KUKA KRL program: MyProgram_065().src

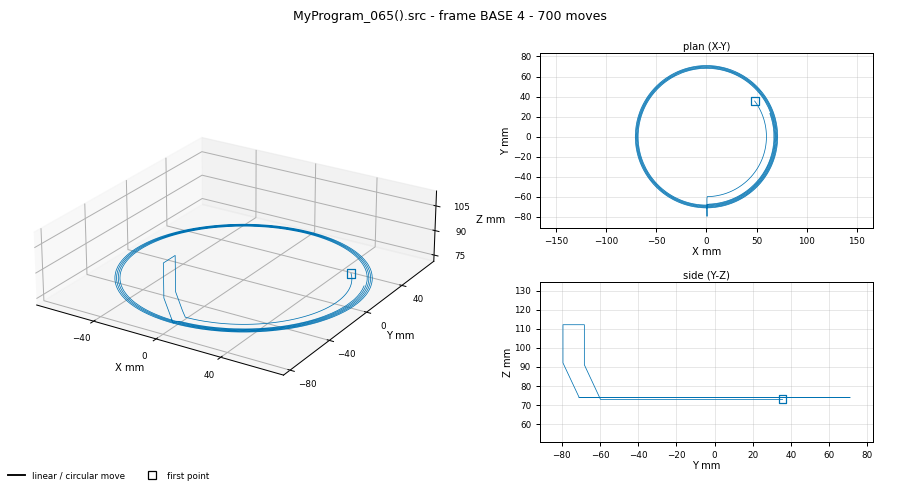
[picture p0: tool path of MyProgram_065().src in frame BASE 4, 700 of 700 moves have a stored position in this frame; points joined in program order, loops and branches not executed]
&ACCESS RVP
&REL 1
&PARAM TEMPLATE = C:\KRC\Roboter\Template\vorgabe
&PARAM EDITMASK = *
DEF MyProgram_065()
; ---- Setting reference (Base) ----
$BASE = BASE_DATA[4]

; --------------------------
; ---- Setting tool (TCP) ----
$TOOL = TOOL_DATA[3]
; --------------------------

$VEL.CP = VEL_APROX_PRINT
Startdeposition()
$VEL.CP = VEL_PRINT
LIN {X 47.9993,Y 35.5944,Z 73,A 29.5508,B 24.867,C -2.6616,E1 25.1296,E2 54.3214} C_DIS
LIN {X 49.6814,Y 33.206,Z 73,A 26.7608,B 24.8676,C -2.6549,E1 25.134,E2 57.1135} C_DIS
LIN {X 51.2611,Y 30.7113,Z 73,A 23.9498,B 24.8683,C -2.648,E1 25.1381,E2 59.9264} C_DIS
LIN {X 52.7031,Y 28.165,Z 73,A 21.1603,B 24.869,C -2.6409,E1 25.1419,E2 62.7181} C_DIS
LIN {X 54.019,Y 25.5508,Z 73,A 18.3589,B 24.8698,C -2.6333,E1 25.1453,E2 65.5225} C_DIS
LIN {X 55.2106,Y 22.862,Z 73,A 15.5717,B 24.8705,C -2.6261,E1 25.1484,E2 68.3114} C_DIS
LIN {X 56.2606,Y 20.1403,Z 73,A 12.7899,B 24.8713,C -2.6184,E1 25.1511,E2 71.096} C_DIS
LIN {X 57.1824,Y 17.3512,Z 73,A 9.9851,B 24.8721,C -2.6104,E1 25.1535,E2 73.9038} C_DIS
LIN {X 57.9667,Y 14.5172,Z 73,A 7.1908,B 24.8728,C -2.6025,E1 25.1555,E2 76.7007} C_DIS
LIN {X 58.6083,Y 11.6601,Z 73,A 4.4011,B 24.8736,C -2.5944,E1 25.1571,E2 79.4934} C_DIS
LIN {X 59.1091,Y 8.7751,Z 73,A 1.6072,B 24.8744,C -2.586,E1 25.1583,E2 82.2905} C_DIS
LIN {X 59.4694,Y 5.855,Z 73,A -1.1879,B 24.8752,C -2.5779,E1 25.1592,E2 85.0884} C_DIS
LIN {X 59.6848,Y 2.935,Z 73,A -3.9767,B 24.8761,C -2.5695,E1 25.1597,E2 87.8804} C_DIS
LIN {X 59.7559,Y 0.0054,Z 73,A -6.7286,B 24.8768,C -2.562,E1 25.1597,E2 90.6337} C_DIS
LIN {X 59.6838,Y -2.9525,Z 73,A -9.5735,B 24.8777,C -2.5528,E1 25.1595,E2 93.4834} C_DIS
LIN {X 59.4691,Y -5.8582,Z 73,A -12.3571,B 24.8785,C -2.5442,E1 25.1588,E2 96.2709} C_DIS
LIN {X 59.1109,Y -8.7628,Z 73,A -15.1438,B 24.8793,C -2.5358,E1 25.1578,E2 99.061} C_DIS
LIN {X 58.611,Y -11.6459,Z 73,A -17.9348,B 24.8801,C -2.5273,E1 25.1563,E2 101.8557} C_DIS
LIN {X 57.9566,Y -14.5566,Z 73,A -20.7653,B 24.8809,C -2.5191,E1 25.1545,E2 104.6892} C_DIS
LIN {X 57.1775,Y -17.3669,Z 73,A -23.5438,B 24.8817,C -2.5109,E1 25.1524,E2 107.4714} C_DIS
LIN {X 56.2608,Y -20.1398,Z 73,A -26.3255,B 24.8824,C -2.5027,E1 25.1498,E2 110.2566} C_DIS
LIN {X 55.2091,Y -22.8658,Z 73,A -29.1109,B 24.8832,C -2.4946,E1 25.1469,E2 113.0457} C_DIS
LIN {X 54.0255,Y -25.5368,Z 73,A -31.8935,B 24.8839,C -2.4868,E1 25.1437,E2 115.8317} C_DIS
LIN {X 52.7131,Y -28.1462,Z 73,A -34.6833,B 24.8847,C -2.4789,E1 25.1401,E2 118.6255} C_DIS
LIN {X 51.2479,Y -30.7332,Z 73,A -37.5078,B 24.8854,C -2.4714,E1 25.1361,E2 121.4531} C_DIS
LIN {X 49.6819,Y -33.2053,Z 73,A -40.2967,B 24.886,C -2.464,E1 25.1319,E2 124.2455} C_DIS
LIN {X 47.9963,Y -35.5983,Z 73,A -43.0873,B 24.8867,C -2.4568,E1 25.1273,E2 127.0396} C_DIS
LIN {X 46.1955,Y -37.906,Z 73,A -45.8892,B 24.8874,C -2.4496,E1 25.1224,E2 129.8455} C_DIS
LIN {X 44.2702,Y -40.1376,Z 73,A -48.6868,B 24.888,C -2.4432,E1 25.1172,E2 132.6458} C_DIS
LIN {X 42.2524,Y -42.2566,Z 73,A -51.4776,B 24.8886,C -2.4367,E1 25.1118,E2 135.4399} C_DIS
LIN {X 40.133,Y -44.2745,Z 73,A -54.2703,B 24.8891,C -2.4305,E1 25.1061,E2 138.2359} C_DIS
LIN {X 37.9019,Y -46.1988,Z 73,A -57.0803,B 24.8897,C -2.4246,E1 25.1001,E2 141.049} C_DIS
LIN {X 35.5942,Y -47.9994,Z 73,A -59.8738,B 24.8902,C -2.419,E1 25.0939,E2 143.8456} C_DIS
LIN {X 33.2009,Y -49.6849,Z 73,A -62.6695,B 24.8907,C -2.4137,E1 25.0874,E2 146.6443} C_DIS
LIN {X 30.728,Y -51.2511,Z 73,A -65.4647,B 24.8911,C -2.4088,E1 25.0808,E2 149.4424} C_DIS
LIN {X 28.1363,Y -52.7183,Z 73,A -68.3046,B 24.8915,C -2.4042,E1 25.0738,E2 152.2848} C_DIS
LIN {X 25.5294,Y -54.0289,Z 73,A -71.094,B 24.8919,C -2.3999,E1 25.0668,E2 155.0769} C_DIS
LIN {X 22.858,Y -55.2123,Z 73,A -73.8869,B 24.8923,C -2.396,E1 25.0596,E2 157.8725} C_DIS
LIN {X 20.1306,Y -56.2641,Z 73,A -76.6835,B 24.8926,C -2.3925,E1 25.0523,E2 160.6715} C_DIS
LIN {X 17.3549,Y -57.1812,Z 73,A -79.4798,B 24.8929,C -2.3893,E1 25.0449,E2 163.4701} C_DIS
LIN {X 14.236,Y -58.0353,Z 73,A -81.964,B 24.8919,C -2.3996,E1 25.0382,E2 165.926} C_DIS
LIN {X 11.905,Y -58.558,Z 73,A -84.7921,B 24.8932,C -2.3859,E1 25.0304,E2 168.783} C_DIS
LIN {X 9.482,Y -58.9998,Z 73,A -87.2165,B 24.8935,C -2.3827,E1 25.0238,E2 171.2124} C_DIS
LIN {X 6.5815,Y -59.3934,Z 73,A -90.0194,B 24.8936,C -2.3811,E1 25.016,E2 174.017} C_DIS
LIN {X 3.6648,Y -59.6444,Z 73,A -92.8251,B 24.8937,C -2.3798,E1 25.0082,E2 176.8243} C_DIS
LIN {X 0.7394,Y -59.7523,Z 73,A -95.6385,B 24.8938,C -2.3788,E1 25.0003,E2 179.6396} C_DIS
LIN {X 0.7394,Y -59.7523,Z 73,A -95.6385,B 24.8938,C -2.3788,E1 25.0003,E2 179.6396} C_DIS
Enddeposition()
LIN {X 0.4348,Y -61.8654,Z 77.5315,A -95.642,B 24.8937,C -2.3803,E1 25.0003,E2 179.6396} C_DIS
LIN {X 0.4346,Y -68.2047,Z 91.1262,A -95.6159,B 24.8947,C -2.3693,E1 25.0003,E2 179.6396} C_DIS
LIN {X 0.4346,Y -68.2047,Z 112.1262,A -95.9721,B 24.8809,C -2.5192,E1 25.0003,E2 179.6396} C_DIS
LIN {X 0.5159,Y -79.41,Z 112.1262,A -95.1989,B 24.897,C -2.3428,E1 25.0013,E2 179.2856} C_DIS
LIN {X 0.5159,Y -79.41,Z 92.1262,A -94.8598,B 24.9092,C -2.2,E1 25.0013,E2 179.2856} C_DIS
LIN {X 0.477,Y -73.0709,Z 78.5315,A -94.8839,B 24.9084,C -2.2101,E1 25.0013,E2 179.2856} C_DIS
LIN {X 0.464,Y -70.9578,Z 74,A -94.8934,B 24.908,C -2.2142,E1 25.0013,E2 179.2856} C_DIS
Startdeposition()
$VEL.CP = VEL_PRINT
LIN {X 2.6443,Y -70.9112,Z 74,A -92.7808,B 24.9072,C -2.2237,E1 25.0073,E2 177.1508} C_DIS
LIN {X 4.3514,Y -70.8271,Z 74,A -91.2694,B 24.9069,C -2.2277,E1 25.0115,E2 175.6306} C_DIS
LIN {X 6.9554,Y -70.619,Z 74,A -89.2706,B 24.9071,C -2.2259,E1 25.017,E2 173.6371} C_DIS
LIN {X 8.6863,Y -70.427,Z 74,A -87.774,B 24.9068,C -2.2291,E1 25.0212,E2 172.134} C_DIS
LIN {X 11.3047,Y -70.0542,Z 74,A -85.4871,B 24.9063,C -2.2345,E1 25.0276,E2 169.8362} C_DIS
LIN {X 13.8437,Y -69.5972,Z 74,A -83.6548,B 24.9067,C -2.2296,E1 25.0325,E2 168.0178} C_DIS
LIN {X 15.5689,Y -69.2315,Z 74,A -82.2744,B 24.9067,C -2.2298,E1 25.0363,E2 166.6388} C_DIS
LIN {X 17.2735,Y -68.826,Z 74,A -80.8713,B 24.9067,C -2.2309,E1 25.0401,E2 165.2352} C_DIS
LIN {X 18.9643,Y -68.3794,Z 74,A -79.4675,B 24.9065,C -2.2321,E1 25.0439,E2 163.8307} C_DIS
LIN {X 20.6298,Y -67.8955,Z 74,A -78.0653,B 24.9064,C -2.2337,E1 25.0477,E2 162.4271} C_DIS
LIN {X 22.2591,Y -67.3791,Z 74,A -76.3904,B 24.9056,C -2.2433,E1 25.0522,E2 160.7327} C_DIS
LIN {X 24.7544,Y -66.5027,Z 74,A -74.38,B 24.9056,C -2.2427,E1 25.0574,E2 158.7278} C_DIS
LIN {X 27.1854,Y -65.5465,Z 74,A -72.4568,B 24.9058,C -2.2406,E1 25.0624,E2 156.8139} C_DIS
LIN {X 28.7858,Y -64.8596,Z 74,A -71.0302,B 24.9056,C -2.2433,E1 25.066,E2 155.3845} C_DIS
LIN {X 30.3689,Y -64.1336,Z 74,A -69.629,B 24.9054,C -2.2453,E1 25.0696,E2 153.982} C_DIS
LIN {X 31.9047,Y -63.3838,Z 74,A -68.2301,B 24.9052,C -2.2481,E1 25.0731,E2 152.5804} C_DIS
LIN {X 34.0253,Y -62.27,Z 74,A -66.2942,B 24.9049,C -2.2514,E1 25.0779,E2 150.6421} C_DIS
LIN {X 35.7594,Y -61.2915,Z 74,A -64.7504,B 24.9049,C -2.2525,E1 25.0816,E2 149.1003} C_DIS
LIN {X 37.2528,Y -60.3955,Z 74,A -63.3253,B 24.9046,C -2.2556,E1 25.085,E2 147.6722} C_DIS
LIN {X 38.7237,Y -59.4631,Z 74,A -61.6883,B 24.9038,C -2.2646,E1 25.0889,E2 146.0193} C_DIS
LIN {X 40.8597,Y -58.0164,Z 74,A -59.628,B 24.9035,C -2.2682,E1 25.0936,E2 143.9577} C_DIS
LIN {X 42.9675,Y -56.4731,Z 74,A -57.7276,B 24.9036,C -2.2668,E1 25.0978,E2 142.0674} C_DIS
LIN {X 44.3657,Y -55.3812,Z 74,A -56.3504,B 24.9035,C -2.2683,E1 25.1009,E2 140.6916} C_DIS
LIN {X 45.7114,Y -54.2757,Z 74,A -54.951,B 24.9032,C -2.2713,E1 25.1039,E2 139.2908} C_DIS
LIN {X 47.0055,Y -53.1592,Z 74,A -53.5535,B 24.9029,C -2.2749,E1 25.1068,E2 137.8902} C_DIS
LIN {X 48.667,Y -51.6406,Z 74,A -51.643,B 24.9023,C -2.2817,E1 25.1107,E2 135.9713} C_DIS
LIN {X 50.1768,Y -50.1768,Z 74,A -50.0323,B 24.9022,C -2.2833,E1 25.1139,E2 134.3636} C_DIS
LIN {X 51.393,Y -48.9302,Z 74,A -48.6338,B 24.9019,C -2.2865,E1 25.1166,E2 132.9636} C_DIS
LIN {X 52.6,Y -47.6301,Z 74,A -47.233,B 24.9017,C -2.2892,E1 25.1193,E2 131.5625} C_DIS
LIN {X 53.732,Y -46.3496,Z 74,A -45.8371,B 24.9013,C -2.2931,E1 25.1219,E2 130.1637} C_DIS
LIN {X 54.8533,Y -45.017,Z 74,A -44.3866,B 24.9009,C -2.298,E1 25.1244,E2 128.7082} C_DIS
LIN {X 56.4731,Y -42.9675,Z 74,A -42.3421,B 24.9006,C -2.3018,E1 25.128,E2 126.6645} C_DIS
LIN {X 57.5294,Y -41.5422,Z 74,A -40.9663,B 24.9004,C -2.304,E1 25.1302,E2 125.2901} C_DIS
LIN {X 58.5316,Y -40.1178,Z 74,A -39.5688,B 24.9001,C -2.3076,E1 25.1324,E2 123.8908} C_DIS
LIN {X 59.481,Y -38.6966,Z 74,A -38.1726,B 24.8997,C -2.3119,E1 25.1346,E2 122.4915} C_DIS
LIN {X 60.4296,Y -37.1975,Z 74,A -36.7739,B 24.8994,C -2.315,E1 25.1367,E2 121.0926} C_DIS
LIN {X 61.3243,Y -35.7032,Z 74,A -35.3516,B 24.8991,C -2.3195,E1 25.1387,E2 119.6671} C_DIS
LIN {X 62.1665,Y -34.2161,Z 74,A -33.9807,B 24.8987,C -2.3232,E1 25.1406,E2 118.2946} C_DIS
LIN {X 63.0023,Y -32.6512,Z 74,A -32.5819,B 24.8985,C -2.3264,E1 25.1424,E2 116.8956} C_DIS
LIN {X 63.8841,Y -30.8881,Z 74,A -30.7867,B 24.8975,C -2.3369,E1 25.1446,E2 115.0851} C_DIS
LIN {X 64.9856,Y -28.4977,Z 74,A -28.6852,B 24.897,C -2.3426,E1 25.147,E2 112.9817} C_DIS
LIN {X 66.1643,Y -25.6439,Z 74,A -26.3784,B 24.8968,C -2.3448,E1 25.1494,E2 110.6824} C_DIS
LIN {X 66.8126,Y -23.9059,Z 74,A -24.877,B 24.8964,C -2.3494,E1 25.1508,E2 109.1784} C_DIS
LIN {X 67.6196,Y -21.516,Z 74,A -22.8479,B 24.8959,C -2.3555,E1 25.1526,E2 107.1464} C_DIS
LIN {X 68.1528,Y -19.7639,Z 74,A -21.2324,B 24.8951,C -2.364,E1 25.1539,E2 105.5201} C_DIS
LIN {X 68.8418,Y -17.2105,Z 74,A -19.2887,B 24.8951,C -2.3652,E1 25.1553,E2 103.5847} C_DIS
LIN {X 69.2763,Y -15.365,Z 74,A -17.541,B 24.894,C -2.3762,E1 25.1564,E2 101.8211} C_DIS
LIN {X 69.7676,Y -12.9567,Z 74,A -15.5786,B 24.8935,C -2.3818,E1 25.1574,E2 99.857} C_DIS
LIN {X 70.1972,Y -10.3799,Z 74,A -13.7032,B 24.8935,C -2.3818,E1 25.1582,E2 97.9926} C_DIS
LIN {X 70.4716,Y -8.3058,Z 74,A -11.8935,B 24.8928,C -2.3906,E1 25.1588,E2 96.1728} C_DIS
LIN {X 70.7016,Y -6.0558,Z 74,A -10.2125,B 24.8926,C -2.3923,E1 25.1593,E2 94.4979} C_DIS
LIN {X 70.8271,Y -4.3514,Z 74,A -8.842,B 24.8922,C -2.3964,E1 25.1595,E2 93.1258} C_DIS
LIN {X 70.9126,Y -2.6119,Z 74,A -7.4223,B 24.8918,C -2.4013,E1 25.1597,E2 91.703} C_DIS
LIN {X 70.9577,Y -0.4157,Z 74,A -5.5996,B 24.8912,C -2.4083,E1 25.1597,E2 89.8745} C_DIS
LIN {X 70.9383,Y 1.7739,Z 74,A -3.9289,B 24.8909,C -2.4111,E1 25.1597,E2 88.2071} C_DIS
LIN {X 70.8734,Y 3.5143,Z 74,A -2.5572,B 24.8906,C -2.4146,E1 25.1595,E2 86.8354} C_DIS
LIN {X 70.7684,Y 5.2202,Z 74,A -1.1383,B 24.8901,C -2.42,E1 25.1593,E2 85.412} C_DIS
LIN {X 70.619,Y 6.9554,Z 74,A 0.2584,B 24.8897,C -2.4242,E1 25.1589,E2 84.0139} C_DIS
LIN {X 70.3476,Y 9.2988,Z 74,A 2.1691,B 24.8892,C -2.4303,E1 25.1583,E2 82.0999} C_DIS
LIN {X 70.0542,Y 11.3047,Z 74,A 3.7266,B 24.8889,C -2.4331,E1 25.1576,E2 80.545} C_DIS
LIN {X 69.7143,Y 13.2353,Z 74,A 5.5384,B 24.8878,C -2.4445,E1 25.1567,E2 78.7169} C_DIS
LIN {X 69.2365,Y 15.5476,Z 74,A 7.2409,B 24.8878,C -2.4445,E1 25.1557,E2 77.0243} C_DIS
LIN {X 68.6498,Y 17.9587,Z 74,A 9.2437,B 24.8873,C -2.4506,E1 25.1543,E2 75.0186} C_DIS
LIN {X 68.1528,Y 19.7639,Z 74,A 10.7329,B 24.8869,C -2.4544,E1 25.1532,E2 73.5289} C_DIS
LIN {X 67.6472,Y 21.4305,Z 74,A 12.1064,B 24.8866,C -2.4577,E1 25.152,E2 72.1555} C_DIS
LIN {X 67.0806,Y 23.142,Z 74,A 13.5311,B 24.8863,C -2.4611,E1 25.1508,E2 70.7308} C_DIS
LIN {X 66.5027,Y 24.7544,Z 74,A 15.0641,B 24.8856,C -2.4693,E1 25.1493,E2 69.1869} C_DIS
LIN {X 65.5465,Y 27.1854,Z 74,A 16.9974,B 24.8855,C -2.4704,E1 25.1473,E2 67.2617} C_DIS
LIN {X 64.7951,Y 28.9289,Z 74,A 18.7915,B 24.8844,C -2.4821,E1 25.1452,E2 65.4498} C_DIS
LIN {X 63.7705,Y 31.1245,Z 74,A 20.49,B 24.8845,C -2.4803,E1 25.1432,E2 63.7647} C_DIS
LIN {X 62.853,Y 32.9355,Z 74,A 22.316,B 24.8836,C -2.49,E1 25.1408,E2 61.9254} C_DIS
LIN {X 61.7419,Y 34.9764,Z 74,A 23.9845,B 24.8837,C -2.4892,E1 25.1386,E2 60.2676} C_DIS
LIN {X 60.5546,Y 36.9917,Z 74,A 25.9115,B 24.8831,C -2.4952,E1 25.1358,E2 58.3362} C_DIS
LIN {X 59.481,Y 38.6966,Z 74,A 27.5132,B 24.8828,C -2.4986,E1 25.1334,E2 56.7344} C_DIS
LIN {X 58.5134,Y 40.1447,Z 74,A 28.8782,B 24.8826,C -2.501,E1 25.1313,E2 55.3706} C_DIS
LIN {X 57.4914,Y 41.5948,Z 74,A 30.3863,B 24.8821,C -2.5067,E1 25.1288,E2 53.8564} C_DIS
LIN {X 55.9416,Y 43.6572,Z 74,A 32.3983,B 24.8818,C -2.5097,E1 25.1254,E2 51.8469} C_DIS
LIN {X 54.5202,Y 45.4178,Z 74,A 34.4814,B 24.8807,C -2.521,E1 25.1217,E2 49.7466} C_DIS
LIN {X 52.5564,Y 47.6782,Z 74,A 36.598,B 24.881,C -2.5181,E1 25.1178,E2 47.6462} C_DIS
LIN {X 51.393,Y 48.9302,Z 74,A 38.2795,B 24.8799,C -2.5294,E1 25.1145,E2 45.9455} C_DIS
LIN {X 49.5158,Y 50.8287,Z 74,A 40.2297,B 24.88,C -2.5282,E1 25.1107,E2 44.0061} C_DIS
LIN {X 47.6543,Y 52.5784,Z 74,A 42.171,B 24.88,C -2.5291,E1 25.1067,E2 42.0708} C_DIS
LIN {X 46.3496,Y 53.732,Z 74,A 43.7638,B 24.8792,C -2.5368,E1 25.1033,E2 40.4659} C_DIS
LIN {X 44.315,Y 55.4218,Z 74,A 45.6976,B 24.8793,C -2.5353,E1 25.0992,E2 38.5429} C_DIS
LIN {X 42.9415,Y 56.4926,Z 74,A 47.0737,B 24.8792,C -2.537,E1 25.0961,E2 37.1678} C_DIS
LIN {X 41.5422,Y 57.5294,Z 74,A 48.7669,B 24.8782,C -2.5471,E1 25.0923,E2 35.4567} C_DIS
LIN {X 39.4236,Y 59.0016,Z 74,A 50.5985,B 24.8785,C -2.5438,E1 25.0881,E2 33.6393} C_DIS
LIN {X 37.9362,Y 59.9686,Z 74,A 52.0025,B 24.8784,C -2.5452,E1 25.0848,E2 32.2364} C_DIS
LIN {X 36.3279,Y 60.9555,Z 74,A 53.7736,B 24.8775,C -2.5541,E1 25.0805,E2 30.4498} C_DIS
LIN {X 34.2161,Y 62.1665,Z 74,A 55.5044,B 24.8779,C -2.5505,E1 25.0763,E2 28.7326} C_DIS
LIN {X 32.6512,Y 63.0023,Z 74,A 57.1456,B 24.8772,C -2.5579,E1 25.0722,E2 27.0785} C_DIS
LIN {X 30.3101,Y 64.1614,Z 74,A 58.9882,B 24.8776,C -2.5534,E1 25.0676,E2 25.2514} C_DIS
LIN {X 28.7048,Y 64.8953,Z 74,A 60.3915,B 24.8776,C -2.5544,E1 25.0641,E2 23.8492} C_DIS
LIN {X 27.1555,Y 65.5591,Z 74,A 62.0198,B 24.8767,C -2.5628,E1 25.0598,E2 22.2047} C_DIS
LIN {X 24.6935,Y 66.5253,Z 74,A 63.8983,B 24.8771,C -2.5582,E1 25.055,E2 20.3413} C_DIS
LIN {X 22.8766,Y 67.1709,Z 74,A 65.6891,B 24.8764,C -2.5656,E1 25.0502,E2 18.5365} C_DIS
LIN {X 20.5676,Y 67.9144,Z 74,A 67.4076,B 24.8769,C -2.5608,E1 25.0457,E2 16.8324} C_DIS
LIN {X 18.8947,Y 68.3987,Z 74,A 68.8116,B 24.8769,C -2.5617,E1 25.0419,E2 15.4286} C_DIS
LIN {X 17.2105,Y 68.8418,Z 74,A 70.3342,B 24.8764,C -2.5656,E1 25.0378,E2 13.8993} C_DIS
LIN {X 14.6649,Y 69.4286,Z 74,A 72.6195,B 24.8759,C -2.5711,E1 25.0315,E2 11.6039} C_DIS
LIN {X 12.1316,Y 69.9159,Z 74,A 74.4535,B 24.8764,C -2.5655,E1 25.0265,E2 9.7851} C_DIS
LIN {X 10.3799,Y 70.1972,Z 74,A 75.8607,B 24.8764,C -2.5653,E1 25.0226,E2 8.3797} C_DIS
LIN {X 8.6863,Y 70.427,Z 74,A 77.4716,B 24.8759,C -2.5714,E1 25.0181,E2 6.7555} C_DIS
LIN {X 6.0558,Y 70.7016,Z 74,A 79.375,B 24.8764,C -2.5658,E1 25.0129,E2 4.8666} C_DIS
LIN {X 4.3514,Y 70.8271,Z 74,A 80.7553,B 24.8764,C -2.5658,E1 25.009,E2 3.4869} C_DIS
LIN {X 2.3084,Y 70.9219,Z 74,A 82.5978,B 24.8759,C -2.5705,E1 25.0039,E2 1.6338} C_DIS
LIN {X -0.456,Y 70.9579,Z 74,A 84.7637,B 24.8761,C -2.5685,E1 24.9978,E2 -0.5271} C_DIS
LIN {X -2.7065,Y 70.9085,Z 74,A 86.413,B 24.8766,C -2.5638,E1 24.9933,E2 -2.1655} C_DIS
LIN {X -5.2202,Y 70.7684,Z 74,A 88.5178,B 24.8766,C -2.5648,E1 24.9874,E2 -4.2732} C_DIS
LIN {X -6.9554,Y 70.619,Z 74,A 90.0917,B 24.8762,C -2.5682,E1 24.983,E2 -5.8561} C_DIS
LIN {X -9.5499,Y 70.3151,Z 74,A 92.0137,B 24.8767,C -2.5624,E1 24.9777,E2 -7.7656} C_DIS
LIN {X -11.3047,Y 70.0542,Z 74,A 93.423,B 24.8769,C -2.5608,E1 24.9738,E2 -9.1726} C_DIS
LIN {X -13.0205,Y 69.7557,Z 74,A 94.832,B 24.8769,C -2.5598,E1 24.9699,E2 -10.5807} C_DIS
LIN {X -14.7285,Y 69.4151,Z 74,A 96.5309,B 24.8764,C -2.5658,E1 24.9652,E2 -12.2957} C_DIS
LIN {X -17.4302,Y 68.7857,Z 74,A 98.7557,B 24.8767,C -2.5633,E1 24.9592,E2 -14.5177} C_DIS
LIN {X -19.7639,Y 68.1528,Z 74,A 100.4914,B 24.8773,C -2.556,E1 24.9546,E2 -16.2388} C_DIS
LIN {X -21.4305,Y 67.6472,Z 74,A 102.0003,B 24.8773,C -2.5569,E1 24.9506,E2 -17.7525} C_DIS
LIN {X -23.9364,Y 66.8015,Z 74,A 104.019,B 24.8778,C -2.5515,E1 24.9453,E2 -19.7622} C_DIS
LIN {X -25.5686,Y 66.1939,Z 74,A 105.4293,B 24.8779,C -2.5498,E1 24.9416,E2 -21.1713} C_DIS
LIN {X -27.1555,Y 65.5591,Z 74,A 106.8194,B 24.8781,C -2.5481,E1 24.938,E2 -22.5606} C_DIS
LIN {X -28.8846,Y 64.8151,Z 74,A 108.5927,B 24.8777,C -2.5519,E1 24.9334,E2 -24.3471} C_DIS
LIN {X -31.1245,Y 63.7705,Z 74,A 110.3407,B 24.8786,C -2.543,E1 24.9291,E2 -26.0784} C_DIS
LIN {X -32.6801,Y 62.9875,Z 74,A 111.776,B 24.8788,C -2.5414,E1 24.9255,E2 -27.5138} C_DIS
LIN {X -34.2161,Y 62.1665,Z 74,A 113.1637,B 24.879,C -2.5386,E1 24.9221,E2 -28.8987} C_DIS
LIN {X -35.7594,Y 61.2915,Z 74,A 114.6641,B 24.8791,C -2.5377,E1 24.9185,E2 -30.4014} C_DIS
LIN {X -37.9638,Y 59.9514,Z 74,A 116.981,B 24.879,C -2.5393,E1 24.9129,E2 -32.7293} C_DIS
LIN {X -40.1447,Y 58.5134,Z 74,A 118.8121,B 24.88,C -2.5288,E1 24.9087,E2 -34.5416} C_DIS
LIN {X -41.5686,Y 57.5106,Z 74,A 120.2486,B 24.8802,C -2.5267,E1 24.9055,E2 -35.978} C_DIS
LIN {X -42.9932,Y 56.4533,Z 74,A 121.6388,B 24.8805,C -2.5228,E1 24.9024,E2 -37.3639} C_DIS
LIN {X -44.4501,Y 55.3127,Z 74,A 123.4197,B 24.8802,C -2.5262,E1 24.8985,E2 -39.1595} C_DIS
LIN {X -46.3496,Y 53.732,Z 74,A 125.1944,B 24.8811,C -2.5168,E1 24.8947,E2 -40.9186} C_DIS
LIN {X -48.2367,Y 52.044,Z 74,A 127.2541,B 24.8815,C -2.5125,E1 24.8905,E2 -42.9763} C_DIS
LIN {X -49.5804,Y 50.7659,Z 74,A 128.7054,B 24.8819,C -2.5079,E1 24.8875,E2 -44.4228} C_DIS
LIN {X -50.8113,Y 49.5338,Z 74,A 130.1192,B 24.8822,C -2.5047,E1 24.8848,E2 -45.8349} C_DIS
LIN {X -52.0269,Y 48.2553,Z 74,A 131.5598,B 24.8825,C -2.5016,E1 24.882,E2 -47.2745} C_DIS
LIN {X -53.1806,Y 46.981,Z 74,A 132.9475,B 24.8829,C -2.4981,E1 24.8794,E2 -48.6601} C_DIS
LIN {X -54.3175,Y 45.6617,Z 74,A 134.6122,B 24.8826,C -2.5004,E1 24.8764,E2 -50.3377} C_DIS
LIN {X -55.9614,Y 43.6315,Z 74,A 136.5084,B 24.8836,C -2.4901,E1 24.8731,E2 -52.2184} C_DIS
LIN {X -57.0153,Y 42.245,Z 74,A 137.9229,B 24.8839,C -2.4866,E1 24.8708,E2 -53.6311} C_DIS
LIN {X -58.0164,Y 40.8597,Z 74,A 139.3355,B 24.8842,C -2.4836,E1 24.8685,E2 -55.0435} C_DIS
LIN {X -59.2957,Y 38.9776,Z 74,A 141.2323,B 24.8846,C -2.4799,E1 24.8655,E2 -56.941} C_DIS
LIN {X -60.6204,Y 36.8835,Z 74,A 143.3221,B 24.8849,C -2.4763,E1 24.8625,E2 -59.0328} C_DIS
LIN {X -61.7419,Y 34.9764,Z 74,A 144.9959,B 24.8856,C -2.4687,E1 24.8601,E2 -60.6972} C_DIS
LIN {X -62.5969,Y 33.4219,Z 74,A 146.4536,B 24.8859,C -2.4651,E1 24.8582,E2 -62.154} C_DIS
LIN {X -63.7561,Y 31.1536,Z 74,A 148.4849,B 24.8866,C -2.4586,E1 24.8557,E2 -64.1806} C_DIS
LIN {X -64.5152,Y 29.5501,Z 74,A 149.9499,B 24.8869,C -2.455,E1 24.8539,E2 -65.6452} C_DIS
LIN {X -65.2209,Y 27.9579,Z 74,A 151.3422,B 24.8873,C -2.4505,E1 24.8524,E2 -67.0344} C_DIS
LIN {X -65.8874,Y 26.3489,Z 74,A 152.7575,B 24.8877,C -2.4465,E1 24.8509,E2 -68.448} C_DIS
LIN {X -66.5142,Y 24.724,Z 74,A 154.4781,B 24.8874,C -2.4491,E1 24.8492,E2 -70.1845} C_DIS
LIN {X -67.3791,Y 22.2591,Z 74,A 156.5959,B 24.888,C -2.4429,E1 24.8473,E2 -72.2995} C_DIS
LIN {X -68.1528,Y 19.7639,Z 74,A 158.4458,B 24.8891,C -2.4307,E1 24.8458,E2 -74.1308} C_DIS
LIN {X -68.7924,Y 17.4041,Z 74,A 160.4541,B 24.8896,C -2.4253,E1 24.8444,E2 -76.138} C_DIS
LIN {X -69.2365,Y 15.5476,Z 74,A 161.9863,B 24.8901,C -2.4202,E1 24.8435,E2 -77.6671} C_DIS
LIN {X -69.5972,Y 13.8437,Z 74,A 163.4022,B 24.8905,C -2.416,E1 24.8427,E2 -79.0813} C_DIS
LIN {X -69.9159,Y 12.1316,Z 74,A 164.8188,B 24.8908,C -2.4118,E1 24.842,E2 -80.4963} C_DIS
LIN {X -70.1972,Y 10.3799,Z 74,A 166.237,B 24.8913,C -2.407,E1 24.8414,E2 -81.9114} C_DIS
LIN {X -70.4408,Y 8.5683,Z 74,A 167.9909,B 24.8911,C -2.4084,E1 24.8407,E2 -83.6792} C_DIS
LIN {X -70.7016,Y 6.0558,Z 74,A 170.0672,B 24.8917,C -2.4027,E1 24.8402,E2 -85.7544} C_DIS
LIN {X -70.8752,Y 3.4819,Z 74,A 171.8763,B 24.8928,C -2.3901,E1 24.8399,E2 -87.5443} C_DIS
LIN {X -70.9472,Y 1.3109,Z 74,A 173.8055,B 24.8929,C -2.3884,E1 24.8398,E2 -89.481} C_DIS
LIN {X -70.9553,Y -0.8708,Z 74,A 175.4408,B 24.8937,C -2.3801,E1 24.8398,E2 -91.1062} C_DIS
LIN {X -70.9112,Y -2.6443,Z 74,A 176.8592,B 24.8941,C -2.3753,E1 24.8399,E2 -92.5216} C_DIS
LIN {X -70.8216,Y -4.4326,Z 74,A 178.5973,B 24.894,C -2.3771,E1 24.8402,E2 -94.2746} C_DIS
LIN {X -70.619,Y -6.9554,Z 74,A -179.602,B 24.895,C -2.3654,E1 24.8407,E2 -96.0581} C_DIS
LIN {X -70.427,Y -8.6863,Z 74,A -178.2105,B 24.8954,C -2.3607,E1 24.8411,E2 -97.4466} C_DIS
LIN {X -70.1926,Y -10.4121,Z 74,A -176.77,B 24.8958,C -2.3571,E1 24.8417,E2 -98.8872} C_DIS
LIN {X -69.9159,Y -12.1316,Z 74,A -175.3542,B 24.8961,C -2.3529,E1 24.8423,E2 -100.3014} C_DIS
LIN {X -69.5972,Y -13.8437,Z 74,A -173.9135,B 24.8964,C -2.3494,E1 24.8431,E2 -101.7422} C_DIS
LIN {X -69.0405,Y -16.396,Z 74,A -171.8138,B 24.897,C -2.3427,E1 24.8444,E2 -103.8384} C_DIS
LIN {X -68.6173,Y -18.0854,Z 74,A -170.3984,B 24.8974,C -2.3387,E1 24.8454,E2 -105.2524} C_DIS
LIN {X -68.1528,Y -19.7639,Z 74,A -168.9827,B 24.8977,C -2.3347,E1 24.8465,E2 -106.6668} C_DIS
LIN {X -67.6472,Y -21.4305,Z 74,A -167.5909,B 24.8981,C -2.3302,E1 24.8476,E2 -108.0559} C_DIS
LIN {X -67.0902,Y -23.1149,Z 74,A -166.1493,B 24.8985,C -2.3263,E1 24.8489,E2 -109.4962} C_DIS
LIN {X -66.5027,Y -24.7544,Z 74,A -164.734,B 24.8988,C -2.3224,E1 24.8503,E2 -110.9102} C_DIS
LIN {X -65.8751,Y -26.379,Z 74,A -163.3185,B 24.8991,C -2.3185,E1 24.8517,E2 -112.3245} C_DIS
LIN {X -65.1132,Y -28.2049,Z 74,A -161.5019,B 24.8991,C -2.3189,E1 24.8537,E2 -114.1521} C_DIS
LIN {X -64.1336,Y -30.3689,Z 74,A -159.7806,B 24.9,C -2.3092,E1 24.8557,E2 -115.8595} C_DIS
LIN {X -63.3838,Y -31.9047,Z 74,A -158.368,B 24.9002,C -2.3061,E1 24.8575,E2 -117.2724} C_DIS
LIN {X -62.5662,Y -33.4792,Z 74,A -156.9756,B 24.9006,C -2.3014,E1 24.8593,E2 -118.6609} C_DIS
LIN {X -61.7419,Y -34.9764,Z 74,A -155.5384,B 24.9008,C -2.299,E1 24.8612,E2 -120.0999} C_DIS
LIN {X -60.5271,Y -37.037,Z 74,A -153.5625,B 24.9012,C -2.295,E1 24.8641,E2 -122.0765} C_DIS
LIN {X -59.4631,Y -38.7237,Z 74,A -152.0249,B 24.9017,C -2.2892,E1 24.8664,E2 -123.6081} C_DIS
LIN {X -58.4949,Y -40.1714,Z 74,A -150.611,B 24.902,C -2.2859,E1 24.8686,E2 -125.0211} C_DIS
LIN {X -57.5106,Y -41.5686,Z 74,A -149.1743,B 24.9021,C -2.2838,E1 24.8709,E2 -126.4598} C_DIS
LIN {X -56.2897,Y -43.2054,Z 74,A -147.3472,B 24.9021,C -2.2839,E1 24.874,E2 -128.296} C_DIS
LIN {X -54.6519,Y -45.2593,Z 74,A -145.2425,B 24.9026,C -2.2786,E1 24.8777,E2 -130.3978} C_DIS
LIN {X -52.9991,Y -47.1843,Z 74,A -143.1263,B 24.9028,C -2.2756,E1 24.8816,E2 -132.5163} C_DIS
LIN {X -51.393,Y -48.9302,Z 74,A -141.4002,B 24.9036,C -2.2671,E1 24.8849,E2 -134.2297} C_DIS
LIN {X -49.9977,Y -50.3537,Z 74,A -139.6104,B 24.9036,C -2.2679,E1 24.8884,E2 -136.0291} C_DIS
LIN {X -48.0838,Y -52.1842,Z 74,A -137.4597,B 24.9038,C -2.2639,E1 24.8928,E2 -138.179} C_DIS
LIN {X -46.2219,Y -53.8408,Z 74,A -135.3977,B 24.9041,C -2.2612,E1 24.8972,E2 -140.2427} C_DIS
LIN {X -44.3404,Y -55.4016,Z 74,A -133.6317,B 24.9048,C -2.2527,E1 24.901,E2 -141.9951} C_DIS
LIN {X -42.9675,Y -56.4731,Z 74,A -132.2201,B 24.905,C -2.2504,E1 24.9041,E2 -143.4063} C_DIS
LIN {X -41.4563,Y -57.5907,Z 74,A -130.4645,B 24.9047,C -2.2535,E1 24.9081,E2 -145.1754} C_DIS
LIN {X -39.4236,Y -59.0016,Z 74,A -128.7155,B 24.9055,C -2.2444,E1 24.9121,E2 -146.9086} C_DIS
LIN {X -37.9638,Y -59.9514,Z 74,A -127.2804,B 24.9056,C -2.2429,E1 24.9155,E2 -148.3448} C_DIS
LIN {X -36.4811,Y -60.865,Z 74,A -125.8695,B 24.9058,C -2.241,E1 24.9188,E2 -149.7555} C_DIS
LIN {X -34.948,Y -61.7578,Z 74,A -124.3544,B 24.9058,C -2.241,E1 24.9225,E2 -151.275} C_DIS
LIN {X -32.6512,Y -63.0023,Z 74,A -122.1824,B 24.9058,C -2.2398,E1 24.9279,E2 -153.4502} C_DIS
LIN {X -30.3396,Y -64.1477,Z 74,A -120.2522,B 24.9064,C -2.2337,E1 24.9327,E2 -155.3709} C_DIS
LIN {X -28.4602,Y -65.002,Z 74,A -118.3602,B 24.9061,C -2.2374,E1 24.9376,E2 -157.2762} C_DIS
LIN {X -25.5686,Y -66.1939,Z 74,A -116.0493,B 24.9067,C -2.2296,E1 24.9435,E2 -159.5738} C_DIS
LIN {X -23.9059,Y -66.8126,Z 74,A -114.5911,B 24.9067,C -2.229,E1 24.9474,E2 -161.0335} C_DIS
LIN {X -22.2281,Y -67.3891,Z 74,A -113.2051,B 24.907,C -2.2268,E1 24.951,E2 -162.4167} C_DIS
LIN {X -20.5676,Y -67.9144,Z 74,A -111.5889,B 24.9066,C -2.2309,E1 24.9554,E2 -164.0455} C_DIS
LIN {X -18.0854,Y -68.6173,Z 74,A -109.6612,B 24.9071,C -2.2258,E1 24.9605,E2 -165.964} C_DIS
LIN {X -16.0884,Y -69.1115,Z 74,A -107.8369,B 24.9068,C -2.229,E1 24.9655,E2 -167.7985} C_DIS
LIN {X -13.8437,Y -69.5972,Z 74,A -106.1423,B 24.9072,C -2.2242,E1 24.9701,E2 -169.4838} C_DIS
LIN {X -12.1316,Y -69.9159,Z 74,A -104.5613,B 24.9069,C -2.2282,E1 24.9745,E2 -171.0757} C_DIS
LIN {X -9.5177,Y -70.3193,Z 74,A -102.4778,B 24.907,C -2.2264,E1 24.9802,E2 -173.1565} C_DIS
LIN {X -6.9554,Y -70.619,Z 74,A -100.5142,B 24.9073,C -2.2231,E1 24.9857,E2 -175.1136} C_DIS
LIN {X -4.6508,Y -70.8069,Z 74,A -98.6127,B 24.9073,C -2.224,E1 24.991,E2 -177.018} C_DIS
LIN {X -2.6119,Y -70.9126,Z 74,A -96.8204,B 24.9069,C -2.2278,E1 24.996,E2 -178.8198} C_DIS
LIN {X 0,Y -70.9607,Z 74,A -94.9146,B 24.9073,C -2.223,E1 25.0013,E2 -180.7142} C_DIS
LIN {X 0,Y -70.9607,Z 74,A -94.9146,B 24.9073,C -2.223,E1 25.0013,E2 -180.7142} C_DIS
Enddeposition()
LIN {X 0.4641,Y -70.0328,Z 74,A -95.2667,B 24.9075,C -2.2208,E1 25.0003,E2 -180.3569} C_DIS
Startdeposition()
$VEL.CP = VEL_PRINT
LIN {X -2.4508,Y -69.9938,Z 74,A -97.8461,B 24.9079,C -2.2155,E1 24.9931,E2 -177.7648} C_DIS
LIN {X -5.377,Y -69.8296,Z 74,A -100.3598,B 24.9082,C -2.2127,E1 24.986,E2 -175.2433} C_DIS
LIN {X -8.408,Y -69.53,Z 74,A -102.8326,B 24.9081,C -2.2134,E1 24.9792,E2 -172.7708} C_DIS
LIN {X -11.6479,Y -69.0607,Z 74,A -105.4844,B 24.908,C -2.2148,E1 24.9719,E2 -170.1199} C_DIS
LIN {X -14.6848,Y -68.4796,Z 74,A -107.8947,B 24.9077,C -2.2187,E1 24.9653,E2 -167.7161} C_DIS
LIN {X -17.1053,Y -67.9159,Z 74,A -109.9308,B 24.9076,C -2.2197,E1 24.9598,E2 -165.6795} C_DIS
LIN {X -19.4877,Y -67.2714,Z 74,A -112.1849,B 24.9079,C -2.2153,E1 24.9537,E2 -163.4115} C_DIS
LIN {X -22.5435,Y -66.3088,Z 74,A -114.6512,B 24.9075,C -2.221,E1 24.9471,E2 -160.9542} C_DIS
LIN {X -26.0919,Y -64.9951,Z 74,A -117.654,B 24.907,C -2.2261,E1 24.9393,E2 -157.9571} C_DIS
LIN {X -31.0293,Y -62.7872,Z 74,A -122.0871,B 24.9066,C -2.2308,E1 24.9281,E2 -153.5243} C_DIS
LIN {X -33.3534,Y -61.584,Z 74,A -124.3421,B 24.9066,C -2.2308,E1 24.9225,E2 -151.2633} C_DIS
LIN {X -35.9278,Y -60.1194,Z 74,A -126.7841,B 24.9064,C -2.2338,E1 24.9166,E2 -148.821} C_DIS
LIN {X -38.0881,Y -58.7744,Z 74,A -129.039,B 24.9064,C -2.233,E1 24.9113,E2 -146.5569} C_DIS
LIN {X -42.3045,Y -55.8163,Z 74,A -133.5902,B 24.9065,C -2.2325,E1 24.901,E2 -141.9884} C_DIS
LIN {X -45.5617,Y -53.1903,Z 74,A -136.5745,B 24.9051,C -2.2487,E1 24.8946,E2 -139.0313} C_DIS
LIN {X -47.6117,Y -51.3643,Z 74,A -138.7539,B 24.9046,C -2.2546,E1 24.8901,E2 -136.8573} C_DIS
LIN {X -49.5827,Y -49.4642,Z 74,A -141.0875,B 24.9044,C -2.2571,E1 24.8855,E2 -134.5198} C_DIS
LIN {X -51.7907,Y -47.147,Z 74,A -143.594,B 24.9037,C -2.2653,E1 24.8807,E2 -132.0219} C_DIS
LIN {X -53.4529,Y -45.2534,Z 74,A -145.652,B 24.9033,C -2.27,E1 24.877,E2 -129.9658} C_DIS
LIN {X -55.3484,Y -42.9144,Z 74,A -148.1595,B 24.9029,C -2.2748,E1 24.8726,E2 -127.458} C_DIS
LIN {X -57.095,Y -40.5614,Z 74,A -150.6195,B 24.9025,C -2.2792,E1 24.8686,E2 -124.9966} C_DIS
LIN {X -58.7529,Y -38.1216,Z 74,A -152.9961,B 24.902,C -2.2861,E1 24.8649,E2 -122.6245} C_DIS
LIN {X -59.7909,Y -36.4705,Z 74,A -154.5732,B 24.9016,C -2.2906,E1 24.8626,E2 -121.0501} C_DIS
LIN {X -61.667,Y -33.2005,Z 74,A -158.1148,B 24.9017,C -2.2889,E1 24.8577,E2 -117.4859} C_DIS
LIN {X -63.4549,Y -29.64,Z 74,A -160.6474,B 24.8996,C -2.3136,E1 24.8547,E2 -114.9985} C_DIS
LIN {X -64.1892,Y -28.014,Z 74,A -162.4972,B 24.8999,C -2.3092,E1 24.8526,E2 -113.1281} C_DIS
LIN {X -65.2797,Y -25.3705,Z 74,A -164.8262,B 24.8993,C -2.3161,E1 24.8502,E2 -110.8026} C_DIS
LIN {X -66.2568,Y -22.6968,Z 74,A -166.8814,B 24.8982,C -2.3288,E1 24.8482,E2 -108.766} C_DIS
LIN {X -67.6059,Y -18.2888,Z 74,A -171.2379,B 24.8984,C -2.3275,E1 24.8448,E2 -104.3813} C_DIS
LIN {X -68.5556,Y -14.3257,Z 74,A -174.3248,B 24.897,C -2.3429,E1 24.8429,E2 -101.313} C_DIS
LIN {X -69.1112,Y -11.3459,Z 74,A -176.8354,B 24.8964,C -2.3499,E1 24.8417,E2 -98.8042} C_DIS
LIN {X -69.6456,Y -7.385,Z 74,A 179.5393,B 24.8962,C -2.3526,E1 24.8404,E2 -95.1636} C_DIS
LIN {X -69.9079,Y -4.2519,Z 74,A 177.288,B 24.8948,C -2.3674,E1 24.84,E2 -92.9341} C_DIS
LIN {X -70.0184,Y -1.6028,Z 74,A 174.5503,B 24.8953,C -2.3623,E1 24.8398,E2 -90.1678} C_DIS
LIN {X -70.0148,Y 1.7647,Z 74,A 172.1848,B 24.8938,C -2.3792,E1 24.8399,E2 -87.8284} C_DIS
LIN {X -69.8312,Y 5.3568,Z 74,A 169.745,B 24.892,C -2.3991,E1 24.8403,E2 -85.4216} C_DIS
LIN {X -69.6637,Y 7.2123,Z 74,A 167.9312,B 24.8921,C -2.3978,E1 24.8408,E2 -83.5938} C_DIS
LIN {X -69.2838,Y 10.2449,Z 74,A 165.328,B 24.8916,C -2.4035,E1 24.8417,E2 -80.9887} C_DIS
LIN {X -68.8629,Y 12.7705,Z 74,A 163.1925,B 24.8911,C -2.4093,E1 24.8428,E2 -78.8543} C_DIS
LIN {X -68.2619,Y 15.6639,Z 74,A 160.9325,B 24.8901,C -2.4202,E1 24.8441,E2 -76.6071} C_DIS
LIN {X -67.7493,Y 17.7532,Z 74,A 158.5897,B 24.8907,C -2.4134,E1 24.8458,E2 -74.2343} C_DIS
LIN {X -66.3642,Y 22.3792,Z 74,A 155.1901,B 24.8885,C -2.4372,E1 24.8486,E2 -70.8721} C_DIS
LIN {X -65.5539,Y 24.6528,Z 74,A 153.0625,B 24.8883,C -2.44,E1 24.8506,E2 -68.739} C_DIS
LIN {X -64.4864,Y 27.3232,Z 74,A 150.6517,B 24.8877,C -2.4458,E1 24.8532,E2 -66.3288} C_DIS
LIN {X -63.3955,Y 29.7675,Z 74,A 148.7209,B 24.8866,C -2.4578,E1 24.8554,E2 -64.4161} C_DIS
LIN {X -62.5352,Y 31.5363,Z 74,A 146.1172,B 24.8881,C -2.4414,E1 24.8587,E2 -61.7593} C_DIS
LIN {X -61.005,Y 34.4024,Z 74,A 144.3767,B 24.8856,C -2.4685,E1 24.861,E2 -60.0742} C_DIS
LIN {X -59.7624,Y 36.5174,Z 74,A 142.1145,B 24.8856,C -2.4687,E1 24.8643,E2 -57.8009} C_DIS
LIN {X -58.0762,Y 39.1435,Z 74,A 139.5351,B 24.885,C -2.4752,E1 24.8682,E2 -55.2239} C_DIS
LIN {X -55.3105,Y 42.9635,Z 74,A 135.5272,B 24.8844,C -2.4822,E1 24.8749,E2 -51.2135} C_DIS
LIN {X -53.0883,Y 45.6814,Z 74,A 132.8377,B 24.8833,C -2.4935,E1 24.8797,E2 -48.5386} C_DIS
LIN {X -51.3894,Y 47.5844,Z 74,A 130.719,B 24.8829,C -2.4979,E1 24.8836,E2 -46.4212} C_DIS
LIN {X -49.3751,Y 49.6708,Z 74,A 128.174,B 24.8827,C -2.4999,E1 24.8886,E2 -43.87} C_DIS
LIN {X -47.1148,Y 51.8203,Z 74,A 125.7941,B 24.8818,C -2.5095,E1 24.8935,E2 -41.5033} C_DIS
LIN {X -45.2098,Y 53.4901,Z 74,A 123.744,B 24.8813,C -2.5146,E1 24.8978,E2 -39.4573} C_DIS
LIN {X -43.1978,Y 55.1278,Z 74,A 121.5393,B 24.8811,C -2.5173,E1 24.9026,E2 -37.2509} C_DIS
LIN {X -41.0266,Y 56.7627,Z 74,A 119.1742,B 24.8809,C -2.5187,E1 24.908,E2 -34.8806} C_DIS
LIN {X -37.9889,Y 58.8381,Z 74,A 116.6854,B 24.8793,C -2.5361,E1 24.9136,E2 -32.4252} C_DIS
LIN {X -36.4168,Y 59.8236,Z 74,A 114.7216,B 24.88,C -2.5289,E1 24.9184,E2 -30.438} C_DIS
LIN {X -33.7108,Y 61.3902,Z 74,A 112.1319,B 24.8796,C -2.5326,E1 24.9247,E2 -27.8496} C_DIS
LIN {X -29.6605,Y 63.4453,Z 74,A 108.8804,B 24.878,C -2.549,E1 24.9327,E2 -24.6286} C_DIS
LIN {X -27.9914,Y 64.1991,Z 74,A 107.246,B 24.8781,C -2.5481,E1 24.9369,E2 -22.9881} C_DIS
LIN {X -26.0012,Y 65.032,Z 74,A 105.1249,B 24.8787,C -2.5423,E1 24.9424,E2 -20.8486} C_DIS
LIN {X -22.6804,Y 66.2627,Z 74,A 102.58,B 24.8775,C -2.5541,E1 24.949,E2 -18.3265} C_DIS
LIN {X -19.8161,Y 67.1742,Z 74,A 99.2561,B 24.8792,C -2.5369,E1 24.958,E2 -14.9561} C_DIS
LIN {X -15.3302,Y 68.3388,Z 74,A 95.9386,B 24.8778,C -2.5514,E1 24.967,E2 -11.6685} C_DIS
LIN {X -12.5562,Y 68.9014,Z 74,A 93.1186,B 24.8787,C -2.5415,E1 24.9748,E2 -8.8218} C_DIS
LIN {X -7.975,Y 69.5807,Z 74,A 89.8218,B 24.8774,C -2.5553,E1 24.9838,E2 -5.5554} C_DIS
LIN {X -5.0014,Y 69.8577,Z 74,A 87.4822,B 24.8771,C -2.5589,E1 24.9903,E2 -3.2233} C_DIS
LIN {X -2.2264,Y 70.0006,Z 74,A 85.1395,B 24.8771,C -2.558,E1 24.9968,E2 -0.878} C_DIS
LIN {X 0.9729,Y 70.0299,Z 74,A 82.469,B 24.8772,C -2.5572,E1 25.0043,E2 1.7943} C_DIS
LIN {X 3.2481,Y 69.961,Z 74,A 80.5708,B 24.8773,C -2.5564,E1 25.0096,E2 3.6937} C_DIS
LIN {X 6.7966,Y 69.7064,Z 74,A 77.6123,B 24.8774,C -2.555,E1 25.0178,E2 6.6539} C_DIS
LIN {X 10.2131,Y 69.2883,Z 74,A 74.8627,B 24.8774,C -2.556,E1 25.0254,E2 9.3989} C_DIS
LIN {X 13.3011,Y 68.7614,Z 74,A 72.552,B 24.8768,C -2.5613,E1 25.0318,E2 11.6945} C_DIS
LIN {X 16.1062,Y 68.1598,Z 74,A 69.9107,B 24.8777,C -2.5528,E1 25.039,E2 14.3525} C_DIS
LIN {X 19.1074,Y 67.3791,Z 74,A 67.442,B 24.8777,C -2.5528,E1 25.0456,E2 16.817} C_DIS
LIN {X 23.1174,Y 66.1108,Z 74,A 64.086,B 24.8777,C -2.5523,E1 25.0545,E2 20.1681} C_DIS
LIN {X 27.8789,Y 64.2481,Z 74,A 60.259,B 24.8772,C -2.5571,E1 25.0644,E2 23.9749} C_DIS
LIN {X 29.8079,Y 63.3767,Z 74,A 58.1701,B 24.8783,C -2.546,E1 25.0697,E2 26.0849} C_DIS
LIN {X 32.3791,Y 62.1025,Z 74,A 55.8438,B 24.8785,C -2.5436,E1 25.0755,E2 28.4106} C_DIS
LIN {X 34.8017,Y 60.7774,Z 74,A 53.4493,B 24.8792,C -2.537,E1 25.0814,E2 30.8136} C_DIS
LIN {X 37.6187,Y 59.0757,Z 74,A 50.8733,B 24.8792,C -2.536,E1 25.0875,E2 33.3839} C_DIS
LIN {X 40.1137,Y 57.4105,Z 74,A 47.8917,B 24.881,C -2.5183,E1 25.0944,E2 36.3971} C_DIS
LIN {X 43.0406,Y 55.2511,Z 74,A 45.4491,B 24.8801,C -2.5269,E1 25.0998,E2 38.8105} C_DIS
LIN {X 45.1672,Y 53.5264,Z 74,A 43.2449,B 24.8804,C -2.5237,E1 25.1045,E2 41.0139} C_DIS
LIN {X 47.667,Y 51.3136,Z 74,A 40.4487,B 24.8811,C -2.5165,E1 25.1103,E2 43.8157} C_DIS
LIN {X 50.0994,Y 48.9412,Z 74,A 37.6444,B 24.8817,C -2.5101,E1 25.1159,E2 46.6235} C_DIS
LIN {X 52.193,Y 46.7004,Z 74,A 35.4046,B 24.8816,C -2.5117,E1 25.12,E2 48.8495} C_DIS
LIN {X 54.1358,Y 44.4357,Z 74,A 32.7911,B 24.8825,C -2.5015,E1 25.1248,E2 51.4753} C_DIS
LIN {X 55.8871,Y 42.2103,Z 74,A 30.5287,B 24.8829,C -2.4974,E1 25.1286,E2 53.7365} C_DIS
LIN {X 57.4226,Y 40.0962,Z 74,A 28.3967,B 24.8834,C -2.4923,E1 25.1321,E2 55.8702} C_DIS
LIN {X 59.1614,Y 37.4851,Z 74,A 25.9572,B 24.8837,C -2.4892,E1 25.1358,E2 58.3049} C_DIS
LIN {X 60.6111,Y 35.0912,Z 74,A 23.3803,B 24.885,C -2.4754,E1 25.1395,E2 60.9011} C_DIS
LIN {X 62.1653,Y 32.2599,Z 74,A 20.8636,B 24.8853,C -2.4717,E1 25.1428,E2 63.4134} C_DIS
LIN {X 63.5219,Y 29.496,Z 74,A 18.2293,B 24.8863,C -2.4616,E1 25.1459,E2 66.0575} C_DIS
LIN {X 65.0407,Y 25.9789,Z 74,A 15.2718,B 24.8867,C -2.4575,E1 25.1491,E2 69.0085} C_DIS
LIN {X 66.2023,Y 22.8566,Z 74,A 12.5397,B 24.8874,C -2.4493,E1 25.1517,E2 71.7443} C_DIS
LIN {X 67.1011,Y 20.0625,Z 74,A 10.135,B 24.8881,C -2.4421,E1 25.1537,E2 74.1524} C_DIS
LIN {X 67.8626,Y 17.3127,Z 74,A 8.236,B 24.8876,C -2.4471,E1 25.155,E2 76.0287} C_DIS
LIN {X 68.3427,Y 15.3127,Z 74,A 6.259,B 24.8888,C -2.4338,E1 25.1563,E2 78.0257} C_DIS
LIN {X 68.8894,Y 12.6231,Z 74,A 4.0711,B 24.8893,C -2.4285,E1 25.1574,E2 80.2132} C_DIS
LIN {X 69.3802,Y 9.5664,Z 74,A 1.7439,B 24.8895,C -2.4264,E1 25.1584,E2 82.5319} C_DIS
LIN {X 69.6529,Y 7.3155,Z 74,A -0.2707,B 24.8904,C -2.4162,E1 25.1591,E2 84.5588} C_DIS
LIN {X 69.8921,Y 4.493,Z 74,A -2.6052,B 24.8911,C -2.4084,E1 25.1595,E2 86.8977} C_DIS
LIN {X 70.0084,Y 1.9732,Z 74,A -4.7007,B 24.8918,C -2.401,E1 25.1598,E2 88.9982} C_DIS
LIN {X 70.0301,Y -0.965,Z 74,A -7.0732,B 24.8924,C -2.3942,E1 25.1598,E2 91.3726} C_DIS
LIN {X 69.8532,Y -5.0644,Z 74,A -10.8358,B 24.8944,C -2.3723,E1 25.1591,E2 95.1646} C_DIS
LIN {X 69.5297,Y -8.4099,Z 74,A -13.1419,B 24.8941,C -2.3759,E1 25.1584,E2 97.4486} C_DIS
LIN {X 69.1133,Y -11.3334,Z 74,A -15.4242,B 24.8944,C -2.3719,E1 25.1575,E2 99.7268} C_DIS
LIN {X 68.6744,Y -13.747,Z 74,A -17.4908,B 24.8951,C -2.3639,E1 25.1564,E2 101.8003} C_DIS
LIN {X 68.1145,Y -16.2959,Z 74,A -19.604,B 24.8957,C -2.3578,E1 25.1551,E2 103.9156} C_DIS
LIN {X 67.4575,Y -18.8307,Z 74,A -21.7209,B 24.8962,C -2.3519,E1 25.1535,E2 106.0345} C_DIS
LIN {X 66.6008,Y -21.6652,Z 74,A -24,B 24.8965,C -2.3483,E1 25.1516,E2 108.3089} C_DIS
LIN {X 65.6413,Y -24.422,Z 74,A -27.1532,B 24.899,C -2.3199,E1 25.1486,E2 111.5116} C_DIS
LIN {X 64.1517,Y -28.1001,Z 74,A -29.8271,B 24.8985,C -2.3259,E1 25.1457,E2 114.1567} C_DIS
LIN {X 62.8071,Y -30.989,Z 74,A -32.3377,B 24.8989,C -2.3209,E1 25.1427,E2 116.6657} C_DIS
LIN {X 60.5552,Y -35.1875,Z 74,A -36.1768,B 24.8998,C -2.3112,E1 25.1375,E2 120.5075} C_DIS
LIN {X 59.1619,Y -37.4844,Z 74,A -38.4319,B 24.9005,C -2.3034,E1 25.1342,E2 122.7695} C_DIS
LIN {X 57.615,Y -39.8194,Z 74,A -40.6421,B 24.9008,C -2.2994,E1 25.1307,E2 124.9785} C_DIS
LIN {X 55.9622,Y -42.1103,Z 74,A -42.8139,B 24.901,C -2.297,E1 25.1271,E2 127.1454} C_DIS
LIN {X 54.833,Y -43.5708,Z 74,A -44.5,B 24.9018,C -2.2882,E1 25.1242,E2 128.8443} C_DIS
LIN {X 52.947,Y -45.8448,Z 74,A -46.8923,B 24.9022,C -2.2827,E1 25.1199,E2 131.2389} C_DIS
LIN {X 50.9529,Y -48.0506,Z 74,A -49.3232,B 24.9028,C -2.2767,E1 25.1153,E2 133.6732} C_DIS
LIN {X 48.8519,Y -50.1862,Z 74,A -51.7773,B 24.9033,C -2.2707,E1 25.1104,E2 136.1311} C_DIS
LIN {X 46.648,Y -52.24,Z 74,A -54.2102,B 24.9037,C -2.2659,E1 25.1054,E2 138.5655} C_DIS
LIN {X 44.3899,Y -54.1731,Z 74,A -56.6452,B 24.9041,C -2.2604,E1 25.1002,E2 141.0041} C_DIS
LIN {X 42.0755,Y -55.9883,Z 74,A -59.0294,B 24.9045,C -2.2559,E1 25.0949,E2 143.3902} C_DIS
LIN {X 39.5981,Y -57.7684,Z 74,A -61.6037,B 24.9051,C -2.2488,E1 25.089,E2 145.9725} C_DIS
LIN {X 37.0065,Y -59.4607,Z 74,A -63.9983,B 24.9052,C -2.2477,E1 25.0834,E2 148.362} C_DIS
LIN {X 34.6086,Y -60.8884,Z 74,A -66.2879,B 24.9056,C -2.2434,E1 25.0778,E2 150.6548} C_DIS
LIN {X 32.1704,Y -62.211,Z 74,A -68.5466,B 24.9059,C -2.2398,E1 25.0722,E2 152.9155} C_DIS
LIN {X 29.6476,Y -63.4513,Z 74,A -70.7704,B 24.906,C -2.2382,E1 25.0667,E2 155.1374} C_DIS
LIN {X 25.9612,Y -65.0477,Z 74,A -74.1905,B 24.9067,C -2.23,E1 25.0578,E2 158.5689} C_DIS
LIN {X 22.0967,Y -66.4595,Z 74,A -77.8988,B 24.9078,C -2.2169,E1 25.048,E2 162.3008} C_DIS
LIN {X 18.6724,Y -67.5023,Z 74,A -80.3063,B 24.907,C -2.227,E1 25.0416,E2 164.6802} C_DIS
LIN {X 15.4891,Y -68.3023,Z 74,A -83.1997,B 24.9076,C -2.2191,E1 25.0337,E2 167.5882} C_DIS
LIN {X 12.5549,Y -68.9017,Z 74,A -85.434,B 24.9073,C -2.2226,E1 25.0276,E2 169.8116} C_DIS
LIN {X 10.1084,Y -69.3032,Z 74,A -87.5694,B 24.9077,C -2.2184,E1 25.0217,E2 171.9549} C_DIS
LIN {X 6.6539,Y -69.7194,Z 74,A -90.3588,B 24.9077,C -2.2182,E1 25.014,E2 174.7427} C_DIS
LIN {X 3.6493,Y -69.9412,Z 74,A -92.8672,B 24.9079,C -2.2161,E1 25.007,E2 177.2552} C_DIS
LIN {X 0.4641,Y -70.0328,Z 74,A -95.266,B 24.9075,C -2.2205,E1 25.0003,E2 179.6431} C_DIS
Enddeposition()
LIN {X 0.4641,Y -70.0328,Z 74,A -95.266,B 24.9075,C -2.2205,E1 25.0003,E2 179.6431} C_DIS
Startdeposition()
$VEL.CP = VEL_PRINT
LIN {X 1.4483,Y -69.0977,Z 74,A -93.68,B 24.9045,C -2.256,E1 25.005,E2 177.9731} C_DIS
LIN {X 4.335,Y -68.9774,Z 74,A -91.2481,B 24.9044,C -2.2578,E1 25.0118,E2 175.5376} C_DIS
LIN {X 7.2559,Y -68.7308,Z 74,A -88.3311,B 24.9032,C -2.2715,E1 25.0199,E2 172.59} C_DIS
LIN {X 11.2233,Y -68.1955,Z 74,A -85.4522,B 24.904,C -2.2626,E1 25.0278,E2 169.735} C_DIS
LIN {X 14.2987,Y -67.6186,Z 74,A -83.0826,B 24.9043,C -2.259,E1 25.0343,E2 167.3767} C_DIS
LIN {X 18.9099,Y -66.4754,Z 74,A -79.1785,B 24.904,C -2.262,E1 25.0449,E2 163.4713} C_DIS
LIN {X 22.1731,Y -65.459,Z 74,A -75.424,B 24.9017,C -2.2894,E1 25.055,E2 159.6588} C_DIS
LIN {X 25.819,Y -64.1093,Z 74,A -72.8924,B 24.9028,C -2.2756,E1 25.0615,E2 157.1656} C_DIS
LIN {X 28.8611,Y -62.799,Z 74,A -69.9507,B 24.9021,C -2.2849,E1 25.069,E2 154.2092} C_DIS
LIN {X 31.515,Y -61.5091,Z 74,A -67.6294,B 24.902,C -2.2856,E1 25.0748,E2 151.8925} C_DIS
LIN {X 34.2409,Y -60.0348,Z 74,A -65.1054,B 24.9017,C -2.2888,E1 25.0809,E2 149.3683} C_DIS
LIN {X 36.8902,Y -58.4447,Z 74,A -62.8571,B 24.902,C -2.2852,E1 25.0863,E2 147.1355} C_DIS
LIN {X 39.0784,Y -57.0052,Z 74,A -60.3446,B 24.9009,C -2.2986,E1 25.0921,E2 144.5999} C_DIS
LIN {X 41.8171,Y -55.0276,Z 74,A -57.4464,B 24.9001,C -2.307,E1 25.0987,E2 141.6921} C_DIS
LIN {X 44.2523,Y -53.0877,Z 74,A -55.1911,B 24.9004,C -2.3038,E1 25.1035,E2 139.4528} C_DIS
LIN {X 46.3779,Y -51.2425,Z 74,A -52.5976,B 24.8993,C -2.3162,E1 25.109,E2 136.8404} C_DIS
LIN {X 48.7728,Y -48.9679,Z 74,A -49.8644,B 24.8988,C -2.3226,E1 25.1144,E2 134.1036} C_DIS
LIN {X 50.9474,Y -46.7003,Z 74,A -47.5564,B 24.8989,C -2.3209,E1 25.1188,E2 131.8096} C_DIS
LIN {X 52.9639,Y -44.4013,Z 74,A -44.9578,B 24.8982,C -2.3291,E1 25.1236,E2 129.2034} C_DIS
LIN {X 54.705,Y -42.2365,Z 74,A -42.3735,B 24.897,C -2.3429,E1 25.1281,E2 126.5986} C_DIS
LIN {X 56.908,Y -39.2188,Z 74,A -39.4569,B 24.8967,C -2.3463,E1 25.1328,E2 123.6882} C_DIS
LIN {X 58.6514,Y -36.5592,Z 74,A -37.3093,B 24.8972,C -2.3402,E1 25.136,E2 121.5657} C_DIS
LIN {X 60.2411,Y -33.8763,Z 74,A -34.4944,B 24.896,C -2.3539,E1 25.14,E2 118.7331} C_DIS
LIN {X 61.1874,Y -32.1351,Z 74,A -32.6076,B 24.895,C -2.3654,E1 25.1425,E2 116.8289} C_DIS
LIN {X 62.7569,Y -28.9514,Z 74,A -29.9091,B 24.8948,C -2.3673,E1 25.1457,E2 114.1404} C_DIS
LIN {X 63.8008,Y -26.5712,Z 74,A -26.8561,B 24.892,C -2.3989,E1 25.1491,E2 111.0296} C_DIS
LIN {X 65.0704,Y -23.2931,Z 74,A -24.7015,B 24.8931,C -2.3865,E1 25.1511,E2 108.9163} C_DIS
LIN {X 66.5239,Y -18.7388,Z 74,A -20.8043,B 24.8922,C -2.3969,E1 25.1543,E2 105.0167} C_DIS
LIN {X 67.2757,Y -15.8308,Z 74,A -18.3762,B 24.8916,C -2.4029,E1 25.1559,E2 102.5884} C_DIS
LIN {X 67.742,Y -13.6977,Z 74,A -16.1729,B 24.8901,C -2.4197,E1 25.1572,E2 100.3584} C_DIS
LIN {X 68.3942,Y -9.9417,Z 74,A -13.4776,B 24.8904,C -2.4166,E1 25.1583,E2 97.6861} C_DIS
LIN {X 68.7002,Y -7.548,Z 74,A -11.1087,B 24.8889,C -2.4333,E1 25.1591,E2 95.2919} C_DIS
LIN {X 69.0393,Y -3.1927,Z 74,A -7.8898,B 24.8889,C -2.4335,E1 25.1597,E2 92.0916} C_DIS
LIN {X 69.1125,Y -0.0717,Z 74,A -4.8416,B 24.8869,C -2.4546,E1 25.1597,E2 89.0116} C_DIS
LIN {X 68.9903,Y 4.1222,Z 74,A -1.7239,B 24.8869,C -2.4555,E1 25.1594,E2 85.9104} C_DIS
LIN {X 68.7809,Y 6.7771,Z 74,A 0.2864,B 24.8867,C -2.4569,E1 25.1589,E2 83.9087} C_DIS
LIN {X 68.4406,Y 9.6152,Z 74,A 2.9597,B 24.8852,C -2.4728,E1 25.1579,E2 81.2137} C_DIS
LIN {X 67.8564,Y 13.1177,Z 74,A 5.7018,B 24.8849,C -2.4762,E1 25.1565,E2 78.4795} C_DIS
LIN {X 67.2198,Y 16.0674,Z 74,A 7.8484,B 24.8851,C -2.474,E1 25.1552,E2 76.3506} C_DIS
LIN {X 66.55,Y 18.6468,Z 74,A 11.2513,B 24.8814,C -2.5138,E1 25.1526,E2 72.8732} C_DIS
LIN {X 65.4411,Y 22.2272,Z 74,A 13.4906,B 24.8828,C -2.4988,E1 25.1507,E2 70.682} C_DIS
LIN {X 64.261,Y 25.4385,Z 74,A 17.3359,B 24.8794,C -2.535,E1 25.1467,E2 66.7726} C_DIS
LIN {X 62.5928,Y 29.304,Z 74,A 19.5463,B 24.8818,C -2.5093,E1 25.1443,E2 64.6347} C_DIS
LIN {X 61.2978,Y 31.9255,Z 74,A 22.1781,B 24.8806,C -2.5216,E1 25.1409,E2 61.9878} C_DIS
LIN {X 58.4388,Y 36.8996,Z 74,A 26.907,B 24.8795,C -2.5333,E1 25.1342,E2 57.2556} C_DIS
LIN {X 57.1523,Y 38.8611,Z 74,A 29.4936,B 24.8774,C -2.5557,E1 25.1301,E2 54.6289} C_DIS
LIN {X 55.2815,Y 41.4791,Z 74,A 31.5347,B 24.8784,C -2.5451,E1 25.1268,E2 52.6226} C_DIS
LIN {X 53.4389,Y 43.8293,Z 74,A 33.6797,B 24.8787,C -2.542,E1 25.123,E2 50.4949} C_DIS
LIN {X 51.7828,Y 45.7742,Z 74,A 36.0998,B 24.8775,C -2.5549,E1 25.1186,E2 48.0553} C_DIS
LIN {X 49.9099,Y 47.808,Z 74,A 38.3994,B 24.877,C -2.5601,E1 25.1142,E2 45.7534} C_DIS
LIN {X 47.7529,Y 49.963,Z 74,A 41.0047,B 24.8763,C -2.5674,E1 25.1089,E2 43.1417} C_DIS
LIN {X 45.0486,Y 52.4144,Z 74,A 44.1057,B 24.8755,C -2.5752,E1 25.1024,E2 40.0344} C_DIS
LIN {X 42.4239,Y 54.5607,Z 74,A 46.6189,B 24.8758,C -2.5725,E1 25.097,E2 37.5371} C_DIS
LIN {X 39.1939,Y 56.9254,Z 74,A 50.4436,B 24.8739,C -2.5913,E1 25.0882,E2 33.6811} C_DIS
LIN {X 36.2855,Y 58.8219,Z 74,A 53.3477,B 24.8734,C -2.5963,E1 25.0813,E2 30.7744} C_DIS
LIN {X 32.3523,Y 61.0731,Z 74,A 56.4451,B 24.8746,C -2.5843,E1 25.0738,E2 27.7145} C_DIS
LIN {X 30.0172,Y 62.2538,Z 74,A 58.632,B 24.8743,C -2.5874,E1 25.0683,E2 25.5261} C_DIS
LIN {X 27.7998,Y 63.2753,Z 74,A 61.0101,B 24.8732,C -2.5987,E1 25.0622,E2 23.127} C_DIS
LIN {X 23.8351,Y 64.8724,Z 74,A 64.1769,B 24.8738,C -2.5925,E1 25.054,E2 19.9818} C_DIS
LIN {X 20.2876,Y 66.0679,Z 74,A 67.2764,B 24.8736,C -2.5949,E1 25.0458,E2 16.8826} C_DIS
LIN {X 18.3101,Y 66.6437,Z 74,A 69.2125,B 24.8729,C -2.6017,E1 25.0406,E2 14.9334} C_DIS
LIN {X 15.2954,Y 67.3994,Z 74,A 71.6811,B 24.873,C -2.6004,E1 25.0339,E2 12.4714} C_DIS
LIN {X 10.7154,Y 68.2771,Z 74,A 75.6819,B 24.8726,C -2.6052,E1 25.0229,E2 8.4637} C_DIS
LIN {X 7.2309,Y 68.7334,Z 74,A 78.4909,B 24.8728,C -2.6031,E1 25.0151,E2 5.6617} C_DIS
LIN {X 4.1707,Y 68.9876,Z 74,A 80.6867,B 24.8736,C -2.5947,E1 25.009,E2 3.4869} C_DIS
LIN {X 0.2308,Y 69.1125,Z 74,A 84.1966,B 24.8731,C -2.6001,E1 24.9992,E2 -0.0352} C_DIS
LIN {X -3.6216,Y 69.018,Z 74,A 87.4675,B 24.873,C -2.601,E1 24.9901,E2 -3.3088} C_DIS
LIN {X -6.6477,Y 68.7929,Z 74,A 89.9764,B 24.8731,C -2.5997,E1 24.9831,E2 -5.8156} C_DIS
LIN {X -10.7189,Y 68.2766,Z 74,A 93.4147,B 24.8732,C -2.5984,E1 24.9736,E2 -9.2537} C_DIS
LIN {X -15.1301,Y 67.4374,Z 74,A 97.1252,B 24.8736,C -2.595,E1 24.9634,E2 -12.9604} C_DIS
LIN {X -17.2071,Y 66.9364,Z 74,A 99.2218,B 24.873,C -2.601,E1 24.9577,E2 -15.0741} C_DIS
LIN {X -21.5966,Y 65.6526,Z 74,A 102.6797,B 24.8742,C -2.5889,E1 24.9486,E2 -18.5094} C_DIS
LIN {X -24.4992,Y 64.6247,Z 74,A 105.0916,B 24.8748,C -2.5825,E1 24.9423,E2 -20.9107} C_DIS
LIN {X -27.2564,Y 63.5121,Z 74,A 108.0698,B 24.874,C -2.5908,E1 24.9345,E2 -23.9155} C_DIS
LIN {X -29.7713,Y 62.372,Z 74,A 110.5333,B 24.874,C -2.5913,E1 24.9283,E2 -26.3865} C_DIS
LIN {X -35.5028,Y 59.2981,Z 74,A 115.3674,B 24.8761,C -2.5693,E1 24.9166,E2 -31.1823} C_DIS
LIN {X -38.3365,Y 57.5052,Z 74,A 118.2951,B 24.8763,C -2.5674,E1 24.9097,E2 -34.1149} C_DIS
LIN {X -41.5913,Y 55.1972,Z 74,A 121.5038,B 24.8771,C -2.5585,E1 24.9025,E2 -37.3137} C_DIS
LIN {X -43.7276,Y 53.5213,Z 74,A 123.7441,B 24.8776,C -2.5535,E1 24.8976,E2 -39.5502} C_DIS
LIN {X -45.9479,Y 51.6274,Z 74,A 126.7252,B 24.8769,C -2.5605,E1 24.8913,E2 -42.56} C_DIS
LIN {X -49.8789,Y 47.8401,Z 74,A 130.7474,B 24.879,C -2.5387,E1 24.8834,E2 -46.547} C_DIS
LIN {X -51.9247,Y 45.6117,Z 74,A 133.3386,B 24.8794,C -2.5343,E1 24.8786,E2 -49.1392} C_DIS
LIN {X -53.201,Y 44.116,Z 74,A 135.6647,B 24.8784,C -2.5453,E1 24.8744,E2 -51.5025} C_DIS
LIN {X -55.2385,Y 41.5363,Z 74,A 137.6837,B 24.8805,C -2.5227,E1 24.871,E2 -53.4772} C_DIS
LIN {X -57.1409,Y 38.8781,Z 74,A 140.5835,B 24.8808,C -2.5195,E1 24.8664,E2 -56.3835} C_DIS
LIN {X -58.7732,Y 36.3643,Z 74,A 142.6269,B 24.8824,C -2.5031,E1 24.8634,E2 -58.398} C_DIS
LIN {X -60.44,Y 33.5202,Z 74,A 146.1288,B 24.8816,C -2.5119,E1 24.8585,E2 -61.9392} C_DIS
LIN {X -62.2687,Y 29.9862,Z 74,A 149.3819,B 24.8826,C -2.5012,E1 24.8545,E2 -65.1844} C_DIS
LIN {X -63.752,Y 26.6884,Z 74,A 151.829,B 24.8845,C -2.4805,E1 24.8518,E2 -67.5955} C_DIS
LIN {X -64.795,Y 24.0482,Z 74,A 154.1039,B 24.8853,C -2.4717,E1 24.8495,E2 -69.8621} C_DIS
LIN {X -65.6376,Y 21.6429,Z 74,A 156.5028,B 24.8853,C -2.4713,E1 24.8473,E2 -72.2738} C_DIS
LIN {X -66.4426,Y 19.0248,Z 74,A 159.0968,B 24.8853,C -2.4712,E1 24.8453,E2 -74.8825} C_DIS
LIN {X -67.2894,Y 15.7719,Z 74,A 162.2732,B 24.8854,C -2.4708,E1 24.8432,E2 -78.0766} C_DIS
LIN {X -67.9511,Y 12.6242,Z 74,A 164.3029,B 24.8875,C -2.4488,E1 24.8422,E2 -80.0657} C_DIS
LIN {X -68.4401,Y 9.6191,Z 74,A 166.8392,B 24.8882,C -2.4411,E1 24.8411,E2 -82.5987} C_DIS
LIN {X -68.8176,Y 6.38,Z 74,A 170.4224,B 24.8872,C -2.4514,E1 24.8401,E2 -86.228} C_DIS
LIN {X -69.0612,Y 2.6809,Z 74,A 172.5128,B 24.89,C -2.4206,E1 24.8399,E2 -88.2573} C_DIS
LIN {X -69.1018,Y -1.225,Z 74,A 176.4474,B 24.8896,C -2.4252,E1 24.8399,E2 -92.2267} C_DIS
LIN {X -68.9258,Y -5.087,Z 74,A -179.9779,B 24.8898,C -2.4231,E1 24.8406,E2 -95.8178} C_DIS
LIN {X -68.5539,Y -8.771,Z 74,A -178.2667,B 24.8933,C -2.3844,E1 24.8411,E2 -97.4468} C_DIS
LIN {X -67.8067,Y -13.3759,Z 74,A -174.1701,B 24.894,C -2.3773,E1 24.843,E2 -101.5507} C_DIS
LIN {X -67.1373,Y -16.4055,Z 74,A -171.0613,B 24.8936,C -2.3809,E1 24.845,E2 -104.6866} C_DIS
LIN {X -66.25,Y -19.6844,Z 74,A -168.3045,B 24.8945,C -2.3713,E1 24.8471,E2 -107.4362} C_DIS
LIN {X -65.3479,Y -22.5027,Z 74,A -165.4591,B 24.8944,C -2.3726,E1 24.8497,E2 -110.301} C_DIS
LIN {X -63.8588,Y -26.4343,Z 74,A -162.4289,B 24.8961,C -2.3527,E1 24.8528,E2 -113.3005} C_DIS
LIN {X -62.7621,Y -28.9404,Z 74,A -159.5245,B 24.8955,C -2.3603,E1 24.8562,E2 -116.2391} C_DIS
LIN {X -60.6868,Y -33.0708,Z 74,A -155.7146,B 24.8964,C -2.3495,E1 24.8612,E2 -120.0433} C_DIS
LIN {X -58.1442,Y -37.3606,Z 74,A -152.3597,B 24.8989,C -2.3216,E1 24.866,E2 -123.3489} C_DIS
LIN {X -56.5285,Y -39.7648,Z 74,A -149.6007,B 24.8987,C -2.3235,E1 24.8704,E2 -126.126} C_DIS
LIN {X -54.7353,Y -42.1973,Z 74,A -146.5347,B 24.8981,C -2.3301,E1 24.8756,E2 -129.2224} C_DIS
LIN {X -52.6755,Y -44.7422,Z 74,A -144.0983,B 24.8992,C -2.3176,E1 24.88,E2 -131.6402} C_DIS
LIN {X -50.1027,Y -47.6068,Z 74,A -140.4723,B 24.899,C -2.3206,E1 24.887,E2 -135.2891} C_DIS
LIN {X -47.5688,Y -50.1384,Z 74,A -138.0107,B 24.9005,C -2.303,E1 24.8919,E2 -137.719} C_DIS
LIN {X -44.5387,Y -52.8489,Z 74,A -134.8528,B 24.9015,C -2.2917,E1 24.8985,E2 -140.8623} C_DIS
LIN {X -41.7514,Y -55.077,Z 74,A -131.753,B 24.9016,C -2.2897,E1 24.9054,E2 -143.9687} C_DIS
LIN {X -38.9145,Y -57.1162,Z 74,A -128.9983,B 24.9023,C -2.2817,E1 24.9116,E2 -146.7138} C_DIS
LIN {X -36.1161,Y -58.9259,Z 74,A -126.1988,B 24.9026,C -2.2784,E1 24.9183,E2 -149.5143} C_DIS
LIN {X -33.2222,Y -60.6048,Z 74,A -123.4747,B 24.903,C -2.2735,E1 24.9249,E2 -152.2347} C_DIS
LIN {X -30.9049,Y -61.8183,Z 74,A -121.0408,B 24.9027,C -2.2771,E1 24.931,E2 -154.6836} C_DIS
LIN {X -27.0255,Y -63.6099,Z 74,A -117.7294,B 24.9035,C -2.2678,E1 24.9394,E2 -157.9808} C_DIS
LIN {X -23.302,Y -65.0663,Z 74,A -114.599,B 24.9041,C -2.2604,E1 24.9475,E2 -161.1002} C_DIS
LIN {X -20.6318,Y -65.9615,Z 74,A -112.0545,B 24.9039,C -2.2636,E1 24.9543,E2 -163.657} C_DIS
LIN {X -17.6697,Y -66.8167,Z 74,A -109.5587,B 24.9041,C -2.2606,E1 24.961,E2 -166.1495} C_DIS
LIN {X -13.8161,Y -67.7177,Z 74,A -106.0284,B 24.9037,C -2.2652,E1 24.9707,E2 -169.695} C_DIS
LIN {X -10.3126,Y -68.3394,Z 74,A -103.3544,B 24.9044,C -2.2575,E1 24.978,E2 -172.3534} C_DIS
LIN {X -7.6843,Y -68.6851,Z 74,A -101.0628,B 24.9042,C -2.2595,E1 24.9844,E2 -174.6513} C_DIS
LIN {X -3.3127,Y -69.0341,Z 74,A -97.6125,B 24.9046,C -2.2549,E1 24.994,E2 -178.092} C_DIS
LIN {X -0.048,Y -69.1137,Z 74,A -94.7417,B 24.9042,C -2.2595,E1 25.002,E2 -180.9738} C_DIS
LIN {X -0.048,Y -69.1137,Z 74,A -94.7417,B 24.9042,C -2.2595,E1 25.002,E2 -180.9738} C_DIS
Enddeposition()
LIN {X 0.463,Y -68.182,Z 74,A -95.8455,B 24.906,C -2.2384,E1 24.9988,E2 -179.8198} C_DIS
Startdeposition()
$VEL.CP = VEL_PRINT
LIN {X -2.7903,Y -68.1324,Z 74,A -99.2767,B 24.9074,C -2.2214,E1 24.9891,E2 -176.3476} C_DIS
LIN {X -6.775,Y -67.8527,Z 74,A -101.5944,B 24.9054,C -2.2461,E1 24.9828,E2 -174.0875} C_DIS
LIN {X -9.432,Y -67.5341,Z 74,A -104.3007,B 24.9062,C -2.2357,E1 24.9753,E2 -171.3546} C_DIS
LIN {X -12.9411,Y -66.9501,Z 74,A -107.8368,B 24.9072,C -2.2241,E1 24.9655,E2 -167.787} C_DIS
LIN {X -16.7368,Y -66.1039,Z 74,A -109.7606,B 24.9044,C -2.257,E1 24.9605,E2 -165.9387} C_DIS
LIN {X -20.3066,Y -65.0956,Z 74,A -113.265,B 24.905,C -2.2501,E1 24.951,E2 -162.4121} C_DIS
LIN {X -23.0625,Y -64.171,Z 74,A -115.8072,B 24.905,C -2.2498,E1 24.9443,E2 -159.8643} C_DIS
LIN {X -25.807,Y -63.1173,Z 74,A -118.6108,B 24.9055,C -2.2446,E1 24.937,E2 -157.0422} C_DIS
LIN {X -30.7803,Y -60.8476,Z 74,A -122.4412,B 24.9036,C -2.2671,E1 24.9274,E2 -153.2558} C_DIS
LIN {X -32.6772,Y -59.85,Z 74,A -124.6486,B 24.9042,C -2.2603,E1 24.9219,E2 -151.0259} C_DIS
LIN {X -35.353,Y -58.3091,Z 74,A -127.926,B 24.9051,C -2.2488,E1 24.914,E2 -147.7113} C_DIS
LIN {X -38.1044,Y -56.5496,Z 74,A -129.5008,B 24.9026,C -2.279,E1 24.9105,E2 -146.2032} C_DIS
LIN {X -40.4566,Y -54.8916,Z 74,A -132.5554,B 24.9034,C -2.2689,E1 24.9034,E2 -143.1138} C_DIS
LIN {X -43.9523,Y -52.1355,Z 74,A -136.1557,B 24.9026,C -2.2788,E1 24.8956,E2 -139.5235} C_DIS
LIN {X -46.4493,Y -49.9237,Z 74,A -138.911,B 24.902,C -2.2853,E1 24.8899,E2 -136.7727} C_DIS
LIN {X -49.4575,Y -46.945,Z 74,A -142.4313,B 24.9013,C -2.2935,E1 24.883,E2 -133.2571} C_DIS
LIN {X -51.584,Y -44.5981,Z 74,A -145.2293,B 24.9011,C -2.2965,E1 24.8778,E2 -130.4537} C_DIS
LIN {X -54.1222,Y -41.4801,Z 74,A -148.5936,B 24.9003,C -2.3047,E1 24.872,E2 -127.0932} C_DIS
LIN {X -55.8113,Y -39.1789,Z 74,A -151.0511,B 24.8999,C -2.3093,E1 24.868,E2 -124.6346} C_DIS
LIN {X -58.2652,Y -35.4253,Z 74,A -154.2341,B 24.898,C -2.3313,E1 24.8632,E2 -121.4881} C_DIS
LIN {X -60.2493,Y -31.9349,Z 74,A -158.1917,B 24.8983,C -2.3279,E1 24.8578,E2 -117.5016} C_DIS
LIN {X -62.0677,Y -28.2392,Z 74,A -161.3683,B 24.897,C -2.3434,E1 24.8539,E2 -114.3448} C_DIS
LIN {X -62.988,Y -26.1237,Z 74,A -164.6933,B 24.899,C -2.3202,E1 24.8503,E2 -110.9461} C_DIS
LIN {X -64.4376,Y -22.3084,Z 74,A -167.1595,B 24.8964,C -2.3499,E1 24.848,E2 -108.5368} C_DIS
LIN {X -65.5774,Y -18.6923,Z 74,A -170.3519,B 24.8956,C -2.3592,E1 24.8455,E2 -105.3483} C_DIS
LIN {X -66.3933,Y -15.5471,Z 74,A -173.1839,B 24.895,C -2.3654,E1 24.8436,E2 -102.5144} C_DIS
LIN {X -67.0043,Y -12.6597,Z 74,A -176.0091,B 24.895,C -2.366,E1 24.842,E2 -99.6739} C_DIS
LIN {X -67.6552,Y -8.5219,Z 74,A -179.2481,B 24.8935,C -2.3826,E1 24.8408,E2 -96.4552} C_DIS
LIN {X -68.0457,Y -4.4267,Z 74,A 177.6403,B 24.8919,C -2.4005,E1 24.8401,E2 -93.3677} C_DIS
LIN {X -68.187,Y -0.5824,Z 74,A 173.7975,B 24.8921,C -2.3983,E1 24.8398,E2 -89.4964} C_DIS
LIN {X -68.1514,Y 2.2807,Z 74,A 171.3535,B 24.8914,C -2.4051,E1 24.84,E2 -87.0541} C_DIS
LIN {X -67.7849,Y 7.4225,Z 74,A 167.7204,B 24.8889,C -2.433,E1 24.8408,E2 -83.4659} C_DIS
LIN {X -67.0761,Y 12.273,Z 74,A 163.3019,B 24.8883,C -2.4399,E1 24.8427,E2 -79.0376} C_DIS
LIN {X -66.5428,Y 14.8976,Z 74,A 161.2289,B 24.8873,C -2.4506,E1 24.8439,E2 -76.9778} C_DIS
LIN {X -66.1444,Y 16.5792,Z 74,A 159.3214,B 24.8877,C -2.4458,E1 24.8452,E2 -75.0478} C_DIS
LIN {X -65.0828,Y 20.3481,Z 74,A 156.5374,B 24.8858,C -2.4664,E1 24.8473,E2 -72.2967} C_DIS
LIN {X -63.9248,Y 23.7394,Z 74,A 153.4311,B 24.8852,C -2.4736,E1 24.8502,E2 -69.19} C_DIS
LIN {X -62.6907,Y 26.8286,Z 74,A 149.4334,B 24.8867,C -2.4575,E1 24.8545,E2 -65.1316} C_DIS
LIN {X -61.1339,Y 30.2065,Z 74,A 147.7194,B 24.8831,C -2.4955,E1 24.8565,E2 -63.4993} C_DIS
LIN {X -59.5073,Y 33.2967,Z 74,A 144.3146,B 24.8832,C -2.4942,E1 24.861,E2 -60.0733} C_DIS
LIN {X -58.0845,Y 35.7223,Z 74,A 141.8997,B 24.8827,C -2.4998,E1 24.8645,E2 -57.6592} C_DIS
LIN {X -56.3172,Y 38.4478,Z 74,A 138.8607,B 24.8827,C -2.5009,E1 24.8692,E2 -54.6077} C_DIS
LIN {X -54.7863,Y 40.6003,Z 74,A 136.5922,B 24.8821,C -2.5057,E1 24.8729,E2 -52.3399} C_DIS
LIN {X -52.1031,Y 43.9903,Z 74,A 133.5794,B 24.88,C -2.5281,E1 24.8782,E2 -49.3663} C_DIS
LIN {X -48.6632,Y 47.7673,Z 74,A 128.9941,B 24.8796,C -2.5325,E1 24.8869,E2 -44.7713} C_DIS
LIN {X -44.7712,Y 51.4329,Z 74,A 124.595,B 24.8784,C -2.5448,E1 24.8959,E2 -40.3836} C_DIS
LIN {X -42.7485,Y 53.1263,Z 74,A 121.5302,B 24.8797,C -2.5315,E1 24.9026,E2 -37.2757} C_DIS
LIN {X -39.9566,Y 55.2577,Z 74,A 119.2506,B 24.8778,C -2.5518,E1 24.9076,E2 -35.0364} C_DIS
LIN {X -36.4155,Y 57.6524,Z 74,A 115.8712,B 24.8767,C -2.5633,E1 24.9154,E2 -31.6732} C_DIS
LIN {X -34.3617,Y 58.9,Z 74,A 113.4907,B 24.8771,C -2.559,E1 24.9212,E2 -29.2753} C_DIS
LIN {X -31.4301,Y 60.5151,Z 74,A 110.5133,B 24.877,C -2.5601,E1 24.9285,E2 -26.2922} C_DIS
LIN {X -26.5178,Y 62.8219,Z 74,A 106.7274,B 24.8746,C -2.584,E1 24.938,E2 -22.5539} C_DIS
LIN {X -24.8092,Y 63.5162,Z 74,A 104.4993,B 24.8759,C -2.571,E1 24.9439,E2 -20.29} C_DIS
LIN {X -20.9565,Y 64.8892,Z 74,A 100.7622,B 24.8761,C -2.5685,E1 24.9538,E2 -16.5398} C_DIS
LIN {X -16.5003,Y 66.1638,Z 74,A 97.2774,B 24.8749,C -2.5816,E1 24.9631,E2 -13.0808} C_DIS
LIN {X -12.2997,Y 67.0713,Z 74,A 94.0491,B 24.8737,C -2.5934,E1 24.9719,E2 -9.8767} C_DIS
LIN {X -7.7601,Y 67.7466,Z 74,A 89.9433,B 24.8741,C -2.5901,E1 24.9833,E2 -5.7597} C_DIS
LIN {X -5.0642,Y 68.002,Z 74,A 86.5474,B 24.8764,C -2.5654,E1 24.9929,E2 -2.3037} C_DIS
LIN {X -1.2194,Y 68.1784,Z 74,A 84.7752,B 24.8731,C -2.6001,E1 24.9976,E2 -0.6139} C_DIS
LIN {X 2.0237,Y 68.1593,Z 74,A 81.1843,B 24.875,C -2.5803,E1 25.0077,E2 3.0238} C_DIS
LIN {X 5.0116,Y 68.0062,Z 74,A 77.96,B 24.8766,C -2.5636,E1 25.0168,E2 6.2862} C_DIS
LIN {X 9.1495,Y 67.5738,Z 74,A 75.8151,B 24.8736,C -2.5947,E1 25.0226,E2 8.3555} C_DIS
LIN {X 13.7691,Y 66.7847,Z 74,A 71.151,B 24.8754,C -2.5759,E1 25.0355,E2 13.0591} C_DIS
LIN {X 18.2887,Y 65.6918,Z 74,A 67.602,B 24.8748,C -2.5821,E1 25.045,E2 16.5878} C_DIS
LIN {X 21.7999,Y 64.6107,Z 74,A 64.7928,B 24.8744,C -2.5865,E1 25.0525,E2 19.3814} C_DIS
LIN {X 24.8236,Y 63.51,Z 74,A 61.2769,B 24.8766,C -2.5642,E1 25.0617,E2 22.9428} C_DIS
LIN {X 28.4535,Y 61.9703,Z 74,A 58.5672,B 24.8755,C -2.5753,E1 25.0686,E2 25.6195} C_DIS
LIN {X 31.413,Y 60.5242,Z 74,A 55.7447,B 24.876,C -2.5705,E1 25.0756,E2 28.4457} C_DIS
LIN {X 34.069,Y 59.0685,Z 74,A 53.1775,B 24.8764,C -2.5664,E1 25.0819,E2 31.0149} C_DIS
LIN {X 37.182,Y 57.161,Z 74,A 50.1077,B 24.8768,C -2.5617,E1 25.0891,E2 34.0861} C_DIS
LIN {X 40.1492,Y 55.1168,Z 74,A 47.0085,B 24.8775,C -2.5548,E1 25.0962,E2 37.1907} C_DIS
LIN {X 42.6547,Y 53.2023,Z 74,A 44.1641,B 24.8784,C -2.5451,E1 25.1025,E2 40.0475} C_DIS
LIN {X 45.0585,Y 51.1819,Z 74,A 41.4301,B 24.8791,C -2.5375,E1 25.1082,E2 42.7886} C_DIS
LIN {X 48.0033,Y 48.4302,Z 74,A 38.182,B 24.8795,C -2.5341,E1 25.1147,E2 46.0313} C_DIS
LIN {X 50.41,Y 45.9203,Z 74,A 35.0752,B 24.8805,C -2.5229,E1 25.1206,E2 49.1508} C_DIS
LIN {X 52.7419,Y 43.2229,Z 74,A 32.6124,B 24.8799,C -2.5298,E1 25.125,E2 51.5862} C_DIS
LIN {X 54.6759,Y 40.7479,Z 74,A 29.3426,B 24.882,C -2.5071,E1 25.1305,E2 54.894} C_DIS
LIN {X 56.6189,Y 38.0022,Z 74,A 27.2625,B 24.8808,C -2.5195,E1 25.1337,E2 56.9346} C_DIS
LIN {X 58.5639,Y 34.9303,Z 74,A 24.0327,B 24.882,C -2.507,E1 25.1385,E2 60.1776} C_DIS
LIN {X 60.6461,Y 31.1747,Z 74,A 20.8534,B 24.8819,C -2.5086,E1 25.1427,E2 63.3363} C_DIS
LIN {X 61.6637,Y 29.112,Z 74,A 18.1916,B 24.8842,C -2.4839,E1 25.1459,E2 66.0421} C_DIS
LIN {X 63.7471,Y 24.2094,Z 74,A 14.2771,B 24.884,C -2.4861,E1 25.15,E2 69.9299} C_DIS
LIN {X 64.9599,Y 20.7366,Z 74,A 11.0741,B 24.8851,C -2.474,E1 25.1529,E2 73.1434} C_DIS
LIN {X 65.9072,Y 17.4951,Z 74,A 8.2951,B 24.8858,C -2.4671,E1 25.1549,E2 75.9228} C_DIS
LIN {X 66.734,Y 14.0162,Z 74,A 5.4302,B 24.8863,C -2.4617,E1 25.1567,E2 78.7838} C_DIS
LIN {X 67.5011,Y 9.664,Z 74,A 1.2257,B 24.8885,C -2.437,E1 25.1586,E2 83.022} C_DIS
LIN {X 67.9036,Y 6.2355,Z 74,A -1.1462,B 24.8881,C -2.4421,E1 25.1593,E2 85.3677} C_DIS
LIN {X 68.1104,Y 3.3005,Z 74,A -4.3657,B 24.8906,C -2.4143,E1 25.1597,E2 88.6339} C_DIS
LIN {X 68.1893,Y -0.0344,Z 74,A -6.0141,B 24.8886,C -2.4365,E1 25.1597,E2 90.2199} C_DIS
LIN {X 68.0754,Y -3.9451,Z 74,A -9.7586,B 24.8907,C -2.4137,E1 25.1594,E2 93.9962} C_DIS
LIN {X 67.7878,Y -7.3951,Z 74,A -12.2214,B 24.8904,C -2.4165,E1 25.1588,E2 96.4376} C_DIS
LIN {X 67.2314,Y -11.3908,Z 74,A -16.0132,B 24.8924,C -2.3949,E1 25.1572,E2 100.2582} C_DIS
LIN {X 66.5314,Y -14.9505,Z 74,A -18.6911,B 24.8924,C -2.3953,E1 25.1557,E2 102.9194} C_DIS
LIN {X 66.0011,Y -17.1368,Z 74,A -21.2374,B 24.8944,C -2.3717,E1 25.1539,E2 105.5068} C_DIS
LIN {X 64.4971,Y -22.1369,Z 74,A -25.7349,B 24.8959,C -2.3552,E1 25.1501,E2 110.0178} C_DIS
LIN {X 62.5033,Y -27.2603,Z 74,A -29.7043,B 24.8956,C -2.3588,E1 25.1459,E2 113.9569} C_DIS
LIN {X 60.823,Y -30.8287,Z 74,A -32.9824,B 24.8964,C -2.3499,E1 25.1419,E2 117.2382} C_DIS
LIN {X 59.9221,Y -32.5443,Z 74,A -35.6352,B 24.8992,C -2.3179,E1 25.1383,E2 119.9528} C_DIS
LIN {X 57.9589,Y -35.925,Z 74,A -37.597,B 24.8969,C -2.3439,E1 25.1356,E2 121.8433} C_DIS
LIN {X 56.8058,Y -37.7218,Z 74,A -39.7471,B 24.8982,C -2.3293,E1 25.1323,E2 124.017} C_DIS
LIN {X 54.0967,Y -41.5133,Z 74,A -43.9477,B 24.8998,C -2.3113,E1 25.1253,E2 128.2401} C_DIS
LIN {X 51.7096,Y -44.4521,Z 74,A -46.7999,B 24.8998,C -2.3118,E1 25.1202,E2 131.0781} C_DIS
LIN {X 49.7479,Y -46.6363,Z 74,A -49.2407,B 24.9002,C -2.3063,E1 25.1156,E2 133.5209} C_DIS
LIN {X 47.0714,Y -49.3375,Z 74,A -52.7606,B 24.9016,C -2.2902,E1 25.1085,E2 137.0642} C_DIS
LIN {X 45.0125,Y -51.2221,Z 74,A -54.7277,B 24.9012,C -2.2947,E1 25.1045,E2 139.0128} C_DIS
LIN {X 42.7745,Y -53.1053,Z 74,A -57.1966,B 24.9017,C -2.289,E1 25.0991,E2 141.4857} C_DIS
LIN {X 40.443,Y -54.9016,Z 74,A -59.9657,B 24.9028,C -2.2762,E1 25.0929,E2 144.2752} C_DIS
LIN {X 35.887,Y -57.9827,Z 74,A -64.0473,B 24.9024,C -2.2812,E1 25.0834,E2 148.3313} C_DIS
LIN {X 33.8731,Y -59.1812,Z 74,A -66.1515,B 24.903,C -2.2742,E1 25.0783,E2 150.4458} C_DIS
LIN {X 31.4511,Y -60.5041,Z 74,A -68.7051,B 24.9038,C -2.2643,E1 25.072,E2 153.0158} C_DIS
LIN {X 29.0052,Y -61.7134,Z 74,A -71.497,B 24.9052,C -2.248,E1 25.0649,E2 155.8388} C_DIS
LIN {X 26.0635,Y -63.0126,Z 74,A -73.2625,B 24.9035,C -2.2678,E1 25.0605,E2 157.5533} C_DIS
LIN {X 24.4838,Y -63.6429,Z 74,A -75.3186,B 24.905,C -2.25,E1 25.055,E2 159.6471} C_DIS
LIN {X 19.6746,Y -65.29,Z 74,A -78.8392,B 24.9039,C -2.2637,E1 25.0458,E2 163.1284} C_DIS
LIN {X 16.0242,Y -66.2799,Z 74,A -82.7182,B 24.9056,C -2.243,E1 25.0352,E2 167.0506} C_DIS
LIN {X 13.0577,Y -66.9277,Z 74,A -85.7918,B 24.9069,C -2.2281,E1 25.0267,E2 170.156} C_DIS
LIN {X 9.4099,Y -67.5372,Z 74,A -88.0534,B 24.9053,C -2.2466,E1 25.0206,E2 172.3716} C_DIS
LIN {X 5.1568,Y -67.9946,Z 74,A -91.1517,B 24.9045,C -2.2568,E1 25.012,E2 175.4437} C_DIS
LIN {X 2.1815,Y -68.1545,Z 74,A -94.0082,B 24.9053,C -2.2472,E1 25.004,E2 178.322} C_DIS
LIN {X 0.463,Y -68.182,Z 74,A -95.8435,B 24.9061,C -2.2375,E1 24.9988,E2 180.1802} C_DIS
Enddeposition()
LIN {X 0.463,Y -68.182,Z 74,A -95.8435,B 24.9061,C -2.2375,E1 24.9988,E2 180.1802} C_DIS
Startdeposition()
$VEL.CP = VEL_PRINT
LIN {X 2.3289,Y -67.2262,Z 74,A -92.8015,B 24.9017,C -2.2891,E1 25.0076,E2 177.0163} C_DIS
LIN {X 4.8568,Y -67.0912,Z 74,A -89.7788,B 24.8998,C -2.3115,E1 25.0162,E2 173.9418} C_DIS
LIN {X 8.4739,Y -66.7303,Z 74,A -87.9555,B 24.9023,C -2.2818,E1 25.0211,E2 172.1903} C_DIS
LIN {X 11.2335,Y -66.3214,Z 74,A -84.8182,B 24.9005,C -2.3024,E1 25.0298,E2 169.0072} C_DIS
LIN {X 14.4557,Y -65.6945,Z 74,A -82.0927,B 24.9005,C -2.303,E1 25.0373,E2 166.2836} C_DIS
LIN {X 18.5913,Y -64.6463,Z 74,A -78.7998,B 24.9009,C -2.2982,E1 25.0461,E2 163.0074} C_DIS
LIN {X 21.9605,Y -63.5812,Z 74,A -75.533,B 24.9,C -2.3084,E1 25.0548,E2 159.7227} C_DIS
LIN {X 25.0586,Y -62.425,Z 74,A -72.9952,B 24.9003,C -2.3051,E1 25.0614,E2 157.1983} C_DIS
LIN {X 27.6194,Y -61.3342,Z 74,A -70.631,B 24.9,C -2.3085,E1 25.0674,E2 154.8319} C_DIS
LIN {X 31.179,Y -59.6034,Z 74,A -67.1466,B 24.8993,C -2.3168,E1 25.0762,E2 151.337} C_DIS
LIN {X 34.0235,Y -58.0273,Z 74,A -64.8836,B 24.9,C -2.3086,E1 25.0816,E2 149.1002} C_DIS
LIN {X 36.3931,Y -56.5709,Z 74,A -61.9518,B 24.8983,C -2.3277,E1 25.0886,E2 146.1327} C_DIS
LIN {X 39.0829,Y -54.747,Z 74,A -59.1109,B 24.8977,C -2.3351,E1 25.0951,E2 143.284} C_DIS
LIN {X 41.9682,Y -52.5689,Z 74,A -56.3,B 24.8977,C -2.3346,E1 25.1013,E2 140.4847} C_DIS
LIN {X 44.1653,Y -50.7361,Z 74,A -53.2388,B 24.8958,C -2.3566,E1 25.1079,E2 137.3834} C_DIS
LIN {X 47.4427,Y -47.6861,Z 74,A -49.8464,B 24.896,C -2.3544,E1 25.1146,E2 134.0105} C_DIS
LIN {X 49.8829,Y -45.128,Z 74,A -47.0852,B 24.896,C -2.3551,E1 25.1198,E2 131.2595} C_DIS
LIN {X 51.5347,Y -43.2318,Z 74,A -44.8443,B 24.8952,C -2.3633,E1 25.1239,E2 129.0096} C_DIS
LIN {X 53.4883,Y -40.79,Z 74,A -42.0864,B 24.8943,C -2.3728,E1 25.1287,E2 126.2422} C_DIS
LIN {X 56.0755,Y -37.1521,Z 74,A -38.5334,B 24.894,C -2.3765,E1 25.1343,E2 122.6979} C_DIS
LIN {X 58.6503,Y -32.9376,Z 74,A -34.3141,B 24.8929,C -2.3888,E1 25.1403,E2 118.4713} C_DIS
LIN {X 60.1544,Y -30.1036,Z 74,A -31.5945,B 24.8922,C -2.3964,E1 25.1438,E2 115.7481} C_DIS
LIN {X 61.3244,Y -27.6411,Z 74,A -29.4921,B 24.8922,C -2.3973,E1 25.1463,E2 113.6548} C_DIS
LIN {X 62.6143,Y -24.5797,Z 74,A -26.1436,B 24.8901,C -2.42,E1 25.1498,E2 110.2713} C_DIS
LIN {X 63.7422,Y -21.486,Z 74,A -23.2432,B 24.8891,C -2.4312,E1 25.1525,E2 107.3607} C_DIS
LIN {X 65.3269,Y -16.0351,Z 74,A -18.4502,B 24.8878,C -2.4451,E1 25.1559,E2 102.5625} C_DIS
LIN {X 66.2904,Y -11.4195,Z 74,A -15.014,B 24.8881,C -2.4418,E1 25.1577,E2 99.154} C_DIS
LIN {X 66.7561,Y -8.2748,Z 74,A -12.3911,B 24.8875,C -2.4481,E1 25.1587,E2 96.5317} C_DIS
LIN {X 66.9996,Y -5.9834,Z 74,A -10.1754,B 24.8863,C -2.4612,E1 25.1593,E2 94.2981} C_DIS
LIN {X 67.2023,Y -2.9278,Z 74,A -7.3017,B 24.8849,C -2.4768,E1 25.1597,E2 91.4048} C_DIS
LIN {X 67.1404,Y 4.129,Z 74,A -1.6866,B 24.8841,C -2.4849,E1 25.1594,E2 85.8039} C_DIS
LIN {X 66.9913,Y 6.0738,Z 74,A 0.1806,B 24.8831,C -2.4957,E1 25.1589,E2 83.9221} C_DIS
LIN {X 66.5616,Y 9.7127,Z 74,A 3.1606,B 24.8825,C -2.5016,E1 25.1578,E2 80.9459} C_DIS
LIN {X 65.7952,Y 13.9938,Z 74,A 6.5399,B 24.8823,C -2.5041,E1 25.156,E2 77.5803} C_DIS
LIN {X 64.6862,Y 18.4508,Z 74,A 10.29,B 24.8816,C -2.5116,E1 25.1534,E2 73.8342} C_DIS
LIN {X 63.1796,Y 23.0879,Z 74,A 14.3338,B 24.8807,C -2.5208,E1 25.1499,E2 69.7915} C_DIS
Enddeposition()
END
